(* IEC 61131-3 sources: elnaProjects/ElpcLogic/PomarKc7Unchanged/build_USO_ecl (part 2) *)

  (* OPC Init - AI. Стартовая инициализация тэгов _______________________________________________________*)

  (********************************************* Модуль A1-4 ******************************************************)

  AI_T_obmotki_fazy_1_k_HL       := ai.T_obmotki_fazy_1_k.HL;
  AI_T_obmotki_fazy_1_k_LL       := ai.T_obmotki_fazy_1_k.LL;
  AI_T_obmotki_fazy_1_k_newHL    := ai.T_obmotki_fazy_1_k.dHL;
  AI_T_obmotki_fazy_1_k_newLL    := ai.T_obmotki_fazy_1_k.dLL;

  AI_T_aktivnogo_zheleza_statora_1_k_HL        := ai.T_aktivnogo_zheleza_statora_1_k.HL;
  AI_T_aktivnogo_zheleza_statora_1_k_LL        := ai.T_aktivnogo_zheleza_statora_1_k.LL;
  AI_T_aktivnogo_zheleza_statora_1_k_newHL     := ai.T_aktivnogo_zheleza_statora_1_k.dHL;
  AI_T_aktivnogo_zheleza_statora_1_k_newLL     := ai.T_aktivnogo_zheleza_statora_1_k.dLL;

  AI_T_obmotki_fazy_2_k_HL	:= ai.T_obmotki_fazy_2_k.HL;
  AI_T_obmotki_fazy_2_k_LL	:= ai.T_obmotki_fazy_2_k.LL;
  AI_T_obmotki_fazy_2_k_newHL	:= ai.T_obmotki_fazy_2_k.dHL;
  AI_T_obmotki_fazy_2_k_newLL	:= ai.T_obmotki_fazy_2_k.dLL;

  AI_T_aktivnogo_zheleza_statora_2_k_HL       := ai.T_aktivnogo_zheleza_statora_2_k.HL;
  AI_T_aktivnogo_zheleza_statora_2_k_LL       := ai.T_aktivnogo_zheleza_statora_2_k.LL;
  AI_T_aktivnogo_zheleza_statora_2_k_newHL    := ai.T_aktivnogo_zheleza_statora_2_k.dHL;
  AI_T_aktivnogo_zheleza_statora_2_k_newLL    := ai.T_aktivnogo_zheleza_statora_2_k.dLL;

  AI_T_obmotki_fazy_3_k_HL	:= ai.T_obmotki_fazy_3_k.HL;
  AI_T_obmotki_fazy_3_k_LL	:= ai.T_obmotki_fazy_3_k.LL;
  AI_T_obmotki_fazy_3_k_newHL	:= ai.T_obmotki_fazy_3_k.dHL;
  AI_T_obmotki_fazy_3_k_newLL	:= ai.T_obmotki_fazy_3_k.dLL;

  AI_T_aktivnogo_zheleza_statora_3_k_HL	    := ai.T_aktivnogo_zheleza_statora_3_k.HL;
  AI_T_aktivnogo_zheleza_statora_3_k_LL	    := ai.T_aktivnogo_zheleza_statora_3_k.LL;
  AI_T_aktivnogo_zheleza_statora_3_k_newHL    := ai.T_aktivnogo_zheleza_statora_3_k.dHL;
  AI_T_aktivnogo_zheleza_statora_3_k_newLL    := ai.T_aktivnogo_zheleza_statora_3_k.dLL;

  AI_T_masla_v_maslobake_HL	:= ai.T_masla_v_maslobake.HL;
  AI_T_masla_v_maslobake_HW	:= ai.T_masla_v_maslobake.HW;
  AI_T_masla_v_maslobake_LL	:= ai.T_masla_v_maslobake.LL;
  AI_T_masla_v_maslobake_LW	:= ai.T_masla_v_maslobake.LW;
  AI_T_masla_v_maslobake_newHL	:= ai.T_masla_v_maslobake.dHL;
  AI_T_masla_v_maslobake_newHW	:= ai.T_masla_v_maslobake.dHW;
  AI_T_masla_v_maslobake_newLL	:= ai.T_masla_v_maslobake.dLL;
  AI_T_masla_v_maslobake_newLW	:= ai.T_masla_v_maslobake.dLW;

  (********************************************* Модуль A1-5 ******************************************************)
  AI_T_perednego_opornogo_podshipnika_dvigatelia_t1_HA	:= ai.T_perednego_opornogo_podshipnika_dvigatelia_t1.HA;
  AI_T_perednego_opornogo_podshipnika_dvigatelia_t1_HL	:= ai.T_perednego_opornogo_podshipnika_dvigatelia_t1.HL;
  AI_T_perednego_opornogo_podshipnika_dvigatelia_t1_HW	:= ai.T_perednego_opornogo_podshipnika_dvigatelia_t1.HW;
  AI_T_perednego_opornogo_podshipnika_dvigatelia_t1_LL	:= ai.T_perednego_opornogo_podshipnika_dvigatelia_t1.LL;
  AI_T_perednego_opornogo_podshipnika_dvigatelia_t1_newHA	:= ai.T_perednego_opornogo_podshipnika_dvigatelia_t1.dHA;
  AI_T_perednego_opornogo_podshipnika_dvigatelia_t1_newHW	:= ai.T_perednego_opornogo_podshipnika_dvigatelia_t1.dHW;
  AI_T_perednego_opornogo_podshipnika_dvigatelia_t1_newHL	:= ai.T_perednego_opornogo_podshipnika_dvigatelia_t1.dHL;
  AI_T_perednego_opornogo_podshipnika_dvigatelia_t1_newLL	:= ai.T_perednego_opornogo_podshipnika_dvigatelia_t1.dLL;

  AI_T_zadnego_opornogo_podshipnika_dvigatelia_t2_HA	:= ai.T_zadnego_opornogo_podshipnika_dvigatelia_t2.HA;
  AI_T_zadnego_opornogo_podshipnika_dvigatelia_t2_HL	:= ai.T_zadnego_opornogo_podshipnika_dvigatelia_t2.HL;
  AI_T_zadnego_opornogo_podshipnika_dvigatelia_t2_HW	:= ai.T_zadnego_opornogo_podshipnika_dvigatelia_t2.HW;
  AI_T_zadnego_opornogo_podshipnika_dvigatelia_t2_LL	:= ai.T_zadnego_opornogo_podshipnika_dvigatelia_t2.LL;
  AI_T_zadnego_opornogo_podshipnika_dvigatelia_t2_newHA	:= ai.T_zadnego_opornogo_podshipnika_dvigatelia_t2.dHA;
  AI_T_zadnego_opornogo_podshipnika_dvigatelia_t2_newHL	:= ai.T_zadnego_opornogo_podshipnika_dvigatelia_t2.dHL;
  AI_T_zadnego_opornogo_podshipnika_dvigatelia_t2_newHW	:= ai.T_zadnego_opornogo_podshipnika_dvigatelia_t2.dHW;
  AI_T_zadnego_opornogo_podshipnika_dvigatelia_t2_newLL	:= ai.T_zadnego_opornogo_podshipnika_dvigatelia_t2.dLL;

  AI_T_masla_na_slive_perednego_opornogo_podshipnika_dvigatelia_HL	:= ai.T_masla_na_slive_perednego_opornogo_podshipnika_dvigatelia.HL;
  AI_T_masla_na_slive_perednego_opornogo_podshipnika_dvigatelia_LL	:= ai.T_masla_na_slive_perednego_opornogo_podshipnika_dvigatelia.LL;
  AI_T_masla_na_slive_perednego_opornogo_podshipnika_dvigatelia_newHL	:= ai.T_masla_na_slive_perednego_opornogo_podshipnika_dvigatelia.dHL;
  AI_T_masla_na_slive_perednego_opornogo_podshipnika_dvigatelia_newLL	:= ai.T_masla_na_slive_perednego_opornogo_podshipnika_dvigatelia.dLL;

  AI_T_masla_na_slive_zadnego_opornogo_podshipnika_dvigatelia_HL	:= ai.T_masla_na_slive_zadnego_opornogo_podshipnika_dvigatelia.HL;
  AI_T_masla_na_slive_zadnego_opornogo_podshipnika_dvigatelia_LL	:= ai.T_masla_na_slive_zadnego_opornogo_podshipnika_dvigatelia.LL;
  AI_T_masla_na_slive_zadnego_opornogo_podshipnika_dvigatelia_newHL	:= ai.T_masla_na_slive_zadnego_opornogo_podshipnika_dvigatelia.dHL;
  AI_T_masla_na_slive_zadnego_opornogo_podshipnika_dvigatelia_newLL	:= ai.T_masla_na_slive_zadnego_opornogo_podshipnika_dvigatelia.dLL;

  AI_T_podshipnika_reduktora_t1_HA	:= ai.T_podshipnika_reduktora_t1.HA;
  AI_T_podshipnika_reduktora_t1_HL	:= ai.T_podshipnika_reduktora_t1.HL;
  AI_T_podshipnika_reduktora_t1_HW	:= ai.T_podshipnika_reduktora_t1.HW;
  AI_T_podshipnika_reduktora_t1_LL	:= ai.T_podshipnika_reduktora_t1.LL;
  AI_T_podshipnika_reduktora_t1_newHA	:= ai.T_podshipnika_reduktora_t1.dHA;
  AI_T_podshipnika_reduktora_t1_newHL	:= ai.T_podshipnika_reduktora_t1.dHL;
  AI_T_podshipnika_reduktora_t1_newHW	:= ai.T_podshipnika_reduktora_t1.dHW;
  AI_T_podshipnika_reduktora_t1_newLL	:= ai.T_podshipnika_reduktora_t1.dLL;

  AI_T_podshipnika_reduktora_t2_HA	:= ai.T_podshipnika_reduktora_t2.HA;
  AI_T_podshipnika_reduktora_t2_HL	:= ai.T_podshipnika_reduktora_t2.HL;
  AI_T_podshipnika_reduktora_t2_HW	:= ai.T_podshipnika_reduktora_t2.HW;
  AI_T_podshipnika_reduktora_t2_LL	:= ai.T_podshipnika_reduktora_t2.LL;
  AI_T_podshipnika_reduktora_t2_newHA	:= ai.T_podshipnika_reduktora_t2.dHA;
  AI_T_podshipnika_reduktora_t2_newHL	:= ai.T_podshipnika_reduktora_t2.dHL;
  AI_T_podshipnika_reduktora_t2_newHW	:= ai.T_podshipnika_reduktora_t2.dHW;
  AI_T_podshipnika_reduktora_t2_newLL	:= ai.T_podshipnika_reduktora_t2.dLL;

  AI_T_podshipnika_reduktora_t3_HA	:= ai.T_podshipnika_reduktora_t3.HA;
  AI_T_podshipnika_reduktora_t3_HL	:= ai.T_podshipnika_reduktora_t3.HL;
  AI_T_podshipnika_reduktora_t3_HW	:= ai.T_podshipnika_reduktora_t3.HW;
  AI_T_podshipnika_reduktora_t3_LL	:= ai.T_podshipnika_reduktora_t3.LL;
  AI_T_podshipnika_reduktora_t3_newHA	:= ai.T_podshipnika_reduktora_t3.dHA;
  AI_T_podshipnika_reduktora_t3_newHL	:= ai.T_podshipnika_reduktora_t3.dHL;
  AI_T_podshipnika_reduktora_t3_newHW	:= ai.T_podshipnika_reduktora_t3.dHW;
  AI_T_podshipnika_reduktora_t3_newLL	:= ai.T_podshipnika_reduktora_t3.dLL;

  AI_T_podshipnika_reduktora_t4_HA	:= ai.T_podshipnika_reduktora_t4.HA;
  AI_T_podshipnika_reduktora_t4_HL	:= ai.T_podshipnika_reduktora_t4.HL;
  AI_T_podshipnika_reduktora_t4_HW	:= ai.T_podshipnika_reduktora_t4.HW;
  AI_T_podshipnika_reduktora_t4_LL	:= ai.T_podshipnika_reduktora_t4.LL;
  AI_T_podshipnika_reduktora_t4_newHA	:= ai.T_podshipnika_reduktora_t4.dHA;
  AI_T_podshipnika_reduktora_t4_newHL	:= ai.T_podshipnika_reduktora_t4.dHL;
  AI_T_podshipnika_reduktora_t4_newHW	:= ai.T_podshipnika_reduktora_t4.dHW;
  AI_T_podshipnika_reduktora_t4_newLL	:= ai.T_podshipnika_reduktora_t4.dLL;

  (********************************************* Модуль A1-6 ******************************************************)

  AI_T_opornogo_podshipnika_nagnetatelia_t1_HA	:= ai.T_opornogo_podshipnika_nagnetatelia_t1.HA;
  AI_T_opornogo_podshipnika_nagnetatelia_t1_HL	:= ai.T_opornogo_podshipnika_nagnetatelia_t1.HL;
  AI_T_opornogo_podshipnika_nagnetatelia_t1_HW	:= ai.T_opornogo_podshipnika_nagnetatelia_t1.HW;
  AI_T_opornogo_podshipnika_nagnetatelia_t1_LL	:= ai.T_opornogo_podshipnika_nagnetatelia_t1.LL;
  AI_T_opornogo_podshipnika_nagnetatelia_t1_newHA	:= ai.T_opornogo_podshipnika_nagnetatelia_t1.dHA;
  AI_T_opornogo_podshipnika_nagnetatelia_t1_newHL	:= ai.T_opornogo_podshipnika_nagnetatelia_t1.dHL;
  AI_T_opornogo_podshipnika_nagnetatelia_t1_newHW	:= ai.T_opornogo_podshipnika_nagnetatelia_t1.dHW;
  AI_T_opornogo_podshipnika_nagnetatelia_t1_newLL	:= ai.T_opornogo_podshipnika_nagnetatelia_t1.dLL;

  AI_T_opornogo_podshipnika_nagnetatelia_t2_HA	:= ai.T_opornogo_podshipnika_nagnetatelia_t2.HA;
  AI_T_opornogo_podshipnika_nagnetatelia_t2_HL	:= ai.T_opornogo_podshipnika_nagnetatelia_t2.HL;
  AI_T_opornogo_podshipnika_nagnetatelia_t2_HW	:= ai.T_opornogo_podshipnika_nagnetatelia_t2.HW;
  AI_T_opornogo_podshipnika_nagnetatelia_t2_LL	:= ai.T_opornogo_podshipnika_nagnetatelia_t2.LL;
  AI_T_opornogo_podshipnika_nagnetatelia_t2_newHA	:= ai.T_opornogo_podshipnika_nagnetatelia_t2.dHA;
  AI_T_opornogo_podshipnika_nagnetatelia_t2_newHL	:= ai.T_opornogo_podshipnika_nagnetatelia_t2.dHL;
  AI_T_opornogo_podshipnika_nagnetatelia_t2_newHW	:= ai.T_opornogo_podshipnika_nagnetatelia_t2.dHW;
  AI_T_opornogo_podshipnika_nagnetatelia_t2_newLL	:= ai.T_opornogo_podshipnika_nagnetatelia_t2.dLL;

  AI_T_opornogo_podshipnika_nagnetatelia_t3_HA	:= ai.T_opornogo_podshipnika_nagnetatelia_t3.HA;
  AI_T_opornogo_podshipnika_nagnetatelia_t3_HL	:= ai.T_opornogo_podshipnika_nagnetatelia_t3.HL;
  AI_T_opornogo_podshipnika_nagnetatelia_t3_HW	:= ai.T_opornogo_podshipnika_nagnetatelia_t3.HW;
  AI_T_opornogo_podshipnika_nagnetatelia_t3_LL	:= ai.T_opornogo_podshipnika_nagnetatelia_t3.LL;
  AI_T_opornogo_podshipnika_nagnetatelia_t3_newHA	:= ai.T_opornogo_podshipnika_nagnetatelia_t3.dHA;
  AI_T_opornogo_podshipnika_nagnetatelia_t3_newHL	:= ai.T_opornogo_podshipnika_nagnetatelia_t3.dHL;
  AI_T_opornogo_podshipnika_nagnetatelia_t3_newHW	:= ai.T_opornogo_podshipnika_nagnetatelia_t3.dHW;
  AI_T_opornogo_podshipnika_nagnetatelia_t3_newLL	:= ai.T_opornogo_podshipnika_nagnetatelia_t3.dLL;

  AI_T_oporno_upornogo_podshipnika_nagnetatelia_t4_HA	:= ai.T_oporno_upornogo_podshipnika_nagnetatelia_t4.HA;
  AI_T_oporno_upornogo_podshipnika_nagnetatelia_t4_HL	:= ai.T_oporno_upornogo_podshipnika_nagnetatelia_t4.HL;
  AI_T_oporno_upornogo_podshipnika_nagnetatelia_t4_HW	:= ai.T_oporno_upornogo_podshipnika_nagnetatelia_t4.HW;
  AI_T_oporno_upornogo_podshipnika_nagnetatelia_t4_LL	:= ai.T_oporno_upornogo_podshipnika_nagnetatelia_t4.LL;
  AI_T_oporno_upornogo_podshipnika_nagnetatelia_t4_newHA	:= ai.T_oporno_upornogo_podshipnika_nagnetatelia_t4.dHA;
  AI_T_oporno_upornogo_podshipnika_nagnetatelia_t4_newHL	:= ai.T_oporno_upornogo_podshipnika_nagnetatelia_t4.dHL;
  AI_T_oporno_upornogo_podshipnika_nagnetatelia_t4_newHW	:= ai.T_oporno_upornogo_podshipnika_nagnetatelia_t4.dHW;
  AI_T_oporno_upornogo_podshipnika_nagnetatelia_t4_newLL	:= ai.T_oporno_upornogo_podshipnika_nagnetatelia_t4.dLL;

  AI_T_masla_do_AVOM_HL	:= ai.T_masla_do_AVOM.HL;
  AI_T_masla_do_AVOM_LL	:= ai.T_masla_do_AVOM.LL;
  AI_T_masla_do_AVOM_newHL	:= ai.T_masla_do_AVOM.dHL;
  AI_T_masla_do_AVOM_newLL	:= ai.T_masla_do_AVOM.dLL;

  AI_T_masla_posle_AVOM_HL	:= ai.T_masla_posle_AVOM.HL;
  AI_T_masla_posle_AVOM_LL	:= ai.T_masla_posle_AVOM.LL;
  AI_T_masla_posle_AVOM_newHL	:= ai.T_masla_posle_AVOM.dHL;
  AI_T_masla_posle_AVOM_newLL	:= ai.T_masla_posle_AVOM.dLL;

  AI_T_gaz_in_nagnetatelia_HL	          := ai.T_gaz_in_nagnetatelia.HL;
  AI_T_gaz_in_nagnetatelia_LL	          := ai.T_gaz_in_nagnetatelia.LL;
  AI_T_gaz_in_nagnetatelia_newHL	:= ai.T_gaz_in_nagnetatelia.dHL;
  AI_T_gaz_in_nagnetatelia_newLL	:= ai.T_gaz_in_nagnetatelia.dLL;

  AI_T_gaz_out_nagnetatelia_HA	          := ai.T_gaz_out_nagnetatelia.HA;
  AI_T_gaz_out_nagnetatelia_HL	          := ai.T_gaz_out_nagnetatelia.HL;
  AI_T_gaz_out_nagnetatelia_HW	          := ai.T_gaz_out_nagnetatelia.HW;
  AI_T_gaz_out_nagnetatelia_LL	          := ai.T_gaz_out_nagnetatelia.LL;
  AI_T_gaz_out_nagnetatelia_newHA	:= ai.T_gaz_out_nagnetatelia.dHA;
  AI_T_gaz_out_nagnetatelia_newHL	:= ai.T_gaz_out_nagnetatelia.dHL;
  AI_T_gaz_out_nagnetatelia_newHW	:= ai.T_gaz_out_nagnetatelia.dHW;
  AI_T_gaz_out_nagnetatelia_newLL	:= ai.T_gaz_out_nagnetatelia.dLL;

  (********************************************* Модуль A1-7 ******************************************************)

  AI_T_clodAir_dvigatelia_t1_HL	          := ai.T_clodAir_dvigatelia_t1.HL;
  AI_T_clodAir_dvigatelia_t1_LL	          := ai.T_clodAir_dvigatelia_t1.LL;
  AI_T_clodAir_dvigatelia_t1_newHL	:= ai.T_clodAir_dvigatelia_t1.dHL;
  AI_T_clodAir_dvigatelia_t1_newLL	:= ai.T_clodAir_dvigatelia_t1.dLL;

  AI_T_hotAir_dvigatelia_t1_HL	          := ai.T_hotAir_dvigatelia_t1.HL;
  AI_T_hotAir_dvigatelia_t1_LL	          := ai.T_hotAir_dvigatelia_t1.LL;
  AI_T_hotAir_dvigatelia_t1_newHL	:= ai.T_hotAir_dvigatelia_t1.dHL;
  AI_T_hotAir_dvigatelia_t1_newLL	:= ai.T_hotAir_dvigatelia_t1.dLL;

  (********************************************* Модуль A1-8 ******************************************************)

  AI_dPmaslo_gaz_HL	          := ai.dPmaslo_gaz.HL;
  AI_dPmaslo_gaz_LA	          := ai.dPmaslo_gaz.LA;
  AI_dPmaslo_gaz_LL	          := ai.dPmaslo_gaz.LL;
  AI_dPmaslo_gaz_LW	          := ai.dPmaslo_gaz.LW;
  AI_dPmaslo_gaz_newHL	:= ai.dPmaslo_gaz.dHL;
  AI_dPmaslo_gaz_newLA	:= ai.dPmaslo_gaz.dLA;
  AI_dPmaslo_gaz_newLL	:= ai.dPmaslo_gaz.dLL;
  AI_dPmaslo_gaz_newLW	:= ai.dPmaslo_gaz.dLW;
  AI_dPmaslo_gaz_newMaxChangeUP	 := ai.dPmaslo_gaz.dMaxChangeSpeed;
  AI_dPmaslo_gaz_newMaxChangeDown := ai.dPmaslo_gaz.dMaxChangeSpeedDown;

  AI_dP_gaza_na_konfuzore_nagnetatelia_HL	          := ai.dP_gaza_na_konfuzore_nagnetatelia.HL;
  AI_dP_gaza_na_konfuzore_nagnetatelia_LL	          := ai.dP_gaza_na_konfuzore_nagnetatelia.LL;
  AI_dP_gaza_na_konfuzore_nagnetatelia_newHL	:= ai.dP_gaza_na_konfuzore_nagnetatelia.dHL;
  AI_dP_gaza_na_konfuzore_nagnetatelia_newLL	:= ai.dP_gaza_na_konfuzore_nagnetatelia.dLL;

  AI_P_masla_uplotneniia_HL	:= ai.P_masla_uplotneniia.HL;
  AI_P_masla_uplotneniia_LL	:= ai.P_masla_uplotneniia.LL;
  AI_P_masla_uplotneniia_newHL	:= ai.P_masla_uplotneniia.dHL;
  AI_P_masla_uplotneniia_newLL	:= ai.P_masla_uplotneniia.dLL;

  AI_P_gaza_na_vkhode_nagnetatelia_HL	:= ai.P_gaza_na_vkhode_nagnetatelia.HL;
  AI_P_gaza_na_vkhode_nagnetatelia_LL	:= ai.P_gaza_na_vkhode_nagnetatelia.LL;
  AI_P_gaza_na_vkhode_nagnetatelia_newHL	:= ai.P_gaza_na_vkhode_nagnetatelia.dHL;
  AI_P_gaza_na_vkhode_nagnetatelia_newLL	:= ai.P_gaza_na_vkhode_nagnetatelia.dLL;

  AI_P_gaza_na_vykhode_nagnetatelia_HL	:= ai.P_gaza_na_vykhode_nagnetatelia.HL;
  AI_P_gaza_na_vykhode_nagnetatelia_LL	:= ai.P_gaza_na_vykhode_nagnetatelia.LL;
  AI_P_gaza_na_vykhode_nagnetatelia_newHL	:= ai.P_gaza_na_vykhode_nagnetatelia.dHL;
  AI_P_gaza_na_vykhode_nagnetatelia_newLL	:= ai.P_gaza_na_vykhode_nagnetatelia.dLL;

  AI_P_masla_smazki_nizkoe_HL	          := ai.P_masla_smazki_nizkoe.HL;
  AI_P_masla_smazki_nizkoe_LA	          := ai.P_masla_smazki_nizkoe.LA;
  AI_P_masla_smazki_nizkoe_LL	          := ai.P_masla_smazki_nizkoe.LL;
  AI_P_masla_smazki_nizkoe_LW	          := ai.P_masla_smazki_nizkoe.LW;
  AI_P_masla_smazki_nizkoe_newHL	:= ai.P_masla_smazki_nizkoe.dHL;
  AI_P_masla_smazki_nizkoe_newLA	:= ai.P_masla_smazki_nizkoe.dLA;
  AI_P_masla_smazki_nizkoe_newLL	:= ai.P_masla_smazki_nizkoe.dLL;
  AI_P_masla_smazki_nizkoe_newLW	:= ai.P_masla_smazki_nizkoe.dLW;

  AI_P_masla_smazki_srednee_posle_nasosov_HL	:= ai.P_masla_smazki_srednee_posle_nasosov.HL;
  AI_P_masla_smazki_srednee_posle_nasosov_LL	:= ai.P_masla_smazki_srednee_posle_nasosov.LL;
  AI_P_masla_smazki_srednee_posle_nasosov_LW	:= ai.P_masla_smazki_srednee_posle_nasosov.LW;
  AI_P_masla_smazki_srednee_posle_nasosov_newHL	:= ai.P_masla_smazki_srednee_posle_nasosov.dHL;
  AI_P_masla_smazki_srednee_posle_nasosov_newLL	:= ai.P_masla_smazki_srednee_posle_nasosov.dLL;
  AI_P_masla_smazki_srednee_posle_nasosov_newLW	:= ai.P_masla_smazki_srednee_posle_nasosov.dLW;

  (********************************************* Модуль A1-9 ******************************************************)

  AI_Vibratciia_STD_t1_HA	:= ai.Vibratciia_STD_t1.HA;
  AI_Vibratciia_STD_t1_HL	:= ai.Vibratciia_STD_t1.HL;
  AI_Vibratciia_STD_t1_HW	:= ai.Vibratciia_STD_t1.HW;
  AI_Vibratciia_STD_t1_LL	:= ai.Vibratciia_STD_t1.LL;
  AI_Vibratciia_STD_t1_newHA	:= ai.Vibratciia_STD_t1.dHA;
  AI_Vibratciia_STD_t1_newHL	:= ai.Vibratciia_STD_t1.dHL;
  AI_Vibratciia_STD_t1_newHW	:= ai.Vibratciia_STD_t1.dHW;
  AI_Vibratciia_STD_t1_newLL	:= ai.Vibratciia_STD_t1.dLL;

  AI_Vibratciia_STD_t2_HA	:= ai.Vibratciia_STD_t2.HA;
  AI_Vibratciia_STD_t2_HL	:= ai.Vibratciia_STD_t2.HL;
  AI_Vibratciia_STD_t2_HW	:= ai.Vibratciia_STD_t2.HW;
  AI_Vibratciia_STD_t2_LL	:= ai.Vibratciia_STD_t2.LL;
  AI_Vibratciia_STD_t2_newHA	:= ai.Vibratciia_STD_t2.dHA;
  AI_Vibratciia_STD_t2_newHL	:= ai.Vibratciia_STD_t2.dHL;
  AI_Vibratciia_STD_t2_newHW	:= ai.Vibratciia_STD_t2.dHW;
  AI_Vibratciia_STD_t2_newLL	:= ai.Vibratciia_STD_t2.dLL;

  AI_Vibratciia_rotora_nagnetatelia_t1_HA	          := ai.Vibratciia_rotora_nagnetatelia_t1.HA;
  AI_Vibratciia_rotora_nagnetatelia_t1_HL	          := ai.Vibratciia_rotora_nagnetatelia_t1.HL;
  AI_Vibratciia_rotora_nagnetatelia_t1_HW	          := ai.Vibratciia_rotora_nagnetatelia_t1.HW;
  AI_Vibratciia_rotora_nagnetatelia_t1_LL	          := ai.Vibratciia_rotora_nagnetatelia_t1.LL;
  AI_Vibratciia_rotora_nagnetatelia_t1_newHA	:= ai.Vibratciia_rotora_nagnetatelia_t1.dHA;
  AI_Vibratciia_rotora_nagnetatelia_t1_newHL	:= ai.Vibratciia_rotora_nagnetatelia_t1.dHL;
  AI_Vibratciia_rotora_nagnetatelia_t1_newHW	:= ai.Vibratciia_rotora_nagnetatelia_t1.dHW;
  AI_Vibratciia_rotora_nagnetatelia_t1_newLL	:= ai.Vibratciia_rotora_nagnetatelia_t1.dLL;

  AI_Vibratciia_rotora_nagnetatelia_t2_HA	          := ai.Vibratciia_rotora_nagnetatelia_t2.HA;
  AI_Vibratciia_rotora_nagnetatelia_t2_HL        	:= ai.Vibratciia_rotora_nagnetatelia_t2.HL;
  AI_Vibratciia_rotora_nagnetatelia_t2_HW    	:= ai.Vibratciia_rotora_nagnetatelia_t2.HW;
  AI_Vibratciia_rotora_nagnetatelia_t2_LL    	:= ai.Vibratciia_rotora_nagnetatelia_t2.LL;
  AI_Vibratciia_rotora_nagnetatelia_t2_newHA	:= ai.Vibratciia_rotora_nagnetatelia_t2.dHA;
  AI_Vibratciia_rotora_nagnetatelia_t2_newHL	:= ai.Vibratciia_rotora_nagnetatelia_t2.dHL;
  AI_Vibratciia_rotora_nagnetatelia_t2_newHW	:= ai.Vibratciia_rotora_nagnetatelia_t2.dHW;
  AI_Vibratciia_rotora_nagnetatelia_t2_newLL	:= ai.Vibratciia_rotora_nagnetatelia_t2.dLL;

  AI_Vibratciia_rotora_nagnetatelia_t3_HA    	:= ai.Vibratciia_rotora_nagnetatelia_t3.HA;
  AI_Vibratciia_rotora_nagnetatelia_t3_HL    	:= ai.Vibratciia_rotora_nagnetatelia_t3.HL;
  AI_Vibratciia_rotora_nagnetatelia_t3_HW    	:= ai.Vibratciia_rotora_nagnetatelia_t3.HW;
  AI_Vibratciia_rotora_nagnetatelia_t3_LL    	:= ai.Vibratciia_rotora_nagnetatelia_t3.LL;
  AI_Vibratciia_rotora_nagnetatelia_t3_newHA	:= ai.Vibratciia_rotora_nagnetatelia_t3.dHA;
  AI_Vibratciia_rotora_nagnetatelia_t3_newHL	:= ai.Vibratciia_rotora_nagnetatelia_t3.dHL;
  AI_Vibratciia_rotora_nagnetatelia_t3_newHW	:= ai.Vibratciia_rotora_nagnetatelia_t3.dHW;
  AI_Vibratciia_rotora_nagnetatelia_t3_newLL	:= ai.Vibratciia_rotora_nagnetatelia_t3.dLL;

  AI_Vibratciia_rotora_nagnetatelia_t4_HA    	:= ai.Vibratciia_rotora_nagnetatelia_t4.HA;
  AI_Vibratciia_rotora_nagnetatelia_t4_HL    	:= ai.Vibratciia_rotora_nagnetatelia_t4.HL;
  AI_Vibratciia_rotora_nagnetatelia_t4_HW    	:= ai.Vibratciia_rotora_nagnetatelia_t4.HW;
  AI_Vibratciia_rotora_nagnetatelia_t4_LL    	:= ai.Vibratciia_rotora_nagnetatelia_t4.LL;
  AI_Vibratciia_rotora_nagnetatelia_t4_newHA	:= ai.Vibratciia_rotora_nagnetatelia_t4.dHA;
  AI_Vibratciia_rotora_nagnetatelia_t4_newHL	:= ai.Vibratciia_rotora_nagnetatelia_t4.dHL;
  AI_Vibratciia_rotora_nagnetatelia_t4_newHW	:= ai.Vibratciia_rotora_nagnetatelia_t4.dHW;
  AI_Vibratciia_rotora_nagnetatelia_t4_newLL	:= ai.Vibratciia_rotora_nagnetatelia_t4.dLL;

  AI_Osevoi_sdvig_rotora_nagnetatelia_HA    	:= ai.Osevoi_sdvig_rotora_nagnetatelia.HA;
  AI_Osevoi_sdvig_rotora_nagnetatelia_HL    	:= ai.Osevoi_sdvig_rotora_nagnetatelia.HL;
  AI_Osevoi_sdvig_rotora_nagnetatelia_HW    	:= ai.Osevoi_sdvig_rotora_nagnetatelia.HW;
  AI_Osevoi_sdvig_rotora_nagnetatelia_LA    	:= ai.Osevoi_sdvig_rotora_nagnetatelia.LA;
  AI_Osevoi_sdvig_rotora_nagnetatelia_LL    	:= ai.Osevoi_sdvig_rotora_nagnetatelia.LL;
  AI_Osevoi_sdvig_rotora_nagnetatelia_LW    	:= ai.Osevoi_sdvig_rotora_nagnetatelia.LW;
  AI_Osevoi_sdvig_rotora_nagnetatelia_newHA	:= ai.Osevoi_sdvig_rotora_nagnetatelia.dHA;
  AI_Osevoi_sdvig_rotora_nagnetatelia_newHL	:= ai.Osevoi_sdvig_rotora_nagnetatelia.dHL;
  AI_Osevoi_sdvig_rotora_nagnetatelia_newHW	:= ai.Osevoi_sdvig_rotora_nagnetatelia.dHW;
  AI_Osevoi_sdvig_rotora_nagnetatelia_newLA	:= ai.Osevoi_sdvig_rotora_nagnetatelia.dLA;
  AI_Osevoi_sdvig_rotora_nagnetatelia_newLL	:= ai.Osevoi_sdvig_rotora_nagnetatelia.dLL;
  AI_Osevoi_sdvig_rotora_nagnetatelia_newLW	:= ai.Osevoi_sdvig_rotora_nagnetatelia.dLW;

  AI_Uroven_masla_v_maslobake_HL	:= ai.Uroven_masla_v_maslobake.HL;
  AI_Uroven_masla_v_maslobake_HW	:= ai.Uroven_masla_v_maslobake.HW;
  AI_Uroven_masla_v_maslobake_LA	:= ai.Uroven_masla_v_maslobake.LA;
  AI_Uroven_masla_v_maslobake_LL	:= ai.Uroven_masla_v_maslobake.LL;
  AI_Uroven_masla_v_maslobake_LW	:= ai.Uroven_masla_v_maslobake.LW;
  AI_Uroven_masla_v_maslobake_newHL	:= ai.Uroven_masla_v_maslobake.dHL;
  AI_Uroven_masla_v_maslobake_newHW	:= ai.Uroven_masla_v_maslobake.dHW;
  AI_Uroven_masla_v_maslobake_newLA	:= ai.Uroven_masla_v_maslobake.dLA;
  AI_Uroven_masla_v_maslobake_newLL	:= ai.Uroven_masla_v_maslobake.dLL;
  AI_Uroven_masla_v_maslobake_newLW	:= ai.Uroven_masla_v_maslobake.dLW;

  (********************************************* Модуль A1-10 ******************************************************)
  AI_T_vnytri_shkafa_HL	:= ai.T_vnytri_shkafa.HL;
  AI_T_vnytri_shkafa_LL	:= ai.T_vnytri_shkafa.LL;
  AI_T_vnytri_shkafa_HW	:= ai.T_vnytri_shkafa.HW;
  AI_T_vnytri_shkafa_LW	:= ai.T_vnytri_shkafa.LW;
  AI_T_vnytri_shkafa_newHL	:= ai.T_vnytri_shkafa.dHL;
  AI_T_vnytri_shkafa_newHW	:= ai.T_vnytri_shkafa.dHW;
  AI_T_vnytri_shkafa_newLL	:= ai.T_vnytri_shkafa.dLL;
  AI_T_vnytri_shkafa_newLW	:= ai.T_vnytri_shkafa.dLW;

  AI_Tok_vozbuzhdeniia_vozbuditelia_HL	:= ai.Tok_vozbuzhdeniia_vozbuditelia.HL;
  AI_Tok_vozbuzhdeniia_vozbuditelia_LL	:= ai.Tok_vozbuzhdeniia_vozbuditelia.LL;
  AI_Tok_vozbuzhdeniia_vozbuditelia_newHL	:= ai.Tok_vozbuzhdeniia_vozbuditelia.dHL;
  AI_Tok_vozbuzhdeniia_vozbuditelia_newLL	:= ai.Tok_vozbuzhdeniia_vozbuditelia.dLL;

  AI_Tok_statora_elektrodvigatelia_HL	:= ai.Tok_statora_elektrodvigatelia.HL;
  AI_Tok_statora_elektrodvigatelia_LL	:= ai.Tok_statora_elektrodvigatelia.LL;
  AI_Tok_statora_elektrodvigatelia_newHL	:= ai.Tok_statora_elektrodvigatelia.dHL;
  AI_Tok_statora_elektrodvigatelia_newLL	:= ai.Tok_statora_elektrodvigatelia.dLL;

  AI_Aktivnaia_moshchnost_HL	:= ai.Aktivnaia_moshchnost.HL;
  AI_Aktivnaia_moshchnost_LL	:= ai.Aktivnaia_moshchnost.LL;
  AI_Aktivnaia_moshchnost_newHL	:= ai.Aktivnaia_moshchnost.dHL;
  AI_Aktivnaia_moshchnost_newLL	:= ai.Aktivnaia_moshchnost.dLL;

  AI_Reaktivnaia_moshchnost_HL    	:= ai.Reaktivnaia_moshchnost.HL;
  AI_Reaktivnaia_moshchnost_LL    	:= ai.Reaktivnaia_moshchnost.LL;
  AI_Reaktivnaia_moshchnost_newHL	:= ai.Reaktivnaia_moshchnost.dHL;
  AI_Reaktivnaia_moshchnost_newLL	:= ai.Reaktivnaia_moshchnost.dLL;

  AI_VoltageSHU_osnovnoi_vvod_HL	:= ai.VoltageSHU_osnovnoi_vvod.HL;
  AI_VoltageSHU_osnovnoi_vvod_HW	:= ai.VoltageSHU_osnovnoi_vvod.HW;
  AI_VoltageSHU_osnovnoi_vvod_LL	:= ai.VoltageSHU_osnovnoi_vvod.LL;
  AI_VoltageSHU_osnovnoi_vvod_LW	:= ai.VoltageSHU_osnovnoi_vvod.LW;
  AI_VoltageSHU_osnovnoi_vvod_newHL	:= ai.VoltageSHU_osnovnoi_vvod.dHL;
  AI_VoltageSHU_osnovnoi_vvod_newHW	:= ai.VoltageSHU_osnovnoi_vvod.dHW;
  AI_VoltageSHU_osnovnoi_vvod_newLL	:= ai.VoltageSHU_osnovnoi_vvod.dLL;
  AI_VoltageSHU_osnovnoi_vvod_newLW	:= ai.VoltageSHU_osnovnoi_vvod.dLW;

  AI_VoltageSHU_rezervnyi_vvod_HL	:= ai.VoltageSHU_rezervnyi_vvod.HL;
  AI_VoltageSHU_rezervnyi_vvod_HW	:= ai.VoltageSHU_rezervnyi_vvod.HW;
  AI_VoltageSHU_rezervnyi_vvod_LL	:= ai.VoltageSHU_rezervnyi_vvod.LL;
  AI_VoltageSHU_rezervnyi_vvod_LW	:= ai.VoltageSHU_rezervnyi_vvod.LW;
  AI_VoltageSHU_rezervnyi_vvod_newHL	:= ai.VoltageSHU_rezervnyi_vvod.dHL;
  AI_VoltageSHU_rezervnyi_vvod_newHW	:= ai.VoltageSHU_rezervnyi_vvod.dHW;
  AI_VoltageSHU_rezervnyi_vvod_newLL	:= ai.VoltageSHU_rezervnyi_vvod.dLL;
  AI_VoltageSHU_rezervnyi_vvod_newLW	:= ai.VoltageSHU_rezervnyi_vvod.dLW;
END_FUNCTION_BLOCK

FUNCTION_BLOCK OPC_AI_get
  VAR_EXTERNAL
    ai : AiConfig;
    AI_Aktivnaia_moshchnost_HL : LREAL;
    AI_Aktivnaia_moshchnost_LL : LREAL;
    AI_Aktivnaia_moshchnost_command : UINT;
    AI_Aktivnaia_moshchnost_newHL : LREAL;
    AI_Aktivnaia_moshchnost_newLL : LREAL;
    AI_Aktivnaia_moshchnost_status : UDINT;
    AI_Aktivnaia_moshchnost_value : LREAL;
    AI_Osevoi_sdvig_rotora_nagnetatelia_HA : LREAL;
    AI_Osevoi_sdvig_rotora_nagnetatelia_HL : LREAL;
    AI_Osevoi_sdvig_rotora_nagnetatelia_HW : LREAL;
    AI_Osevoi_sdvig_rotora_nagnetatelia_LA : LREAL;
    AI_Osevoi_sdvig_rotora_nagnetatelia_LL : LREAL;
    AI_Osevoi_sdvig_rotora_nagnetatelia_LW : LREAL;
    AI_Osevoi_sdvig_rotora_nagnetatelia_command : UINT;
    AI_Osevoi_sdvig_rotora_nagnetatelia_newHA : LREAL;
    AI_Osevoi_sdvig_rotora_nagnetatelia_newHL : LREAL;
    AI_Osevoi_sdvig_rotora_nagnetatelia_newHW : LREAL;
    AI_Osevoi_sdvig_rotora_nagnetatelia_newLA : LREAL;
    AI_Osevoi_sdvig_rotora_nagnetatelia_newLL : LREAL;
    AI_Osevoi_sdvig_rotora_nagnetatelia_newLW : LREAL;
    AI_Osevoi_sdvig_rotora_nagnetatelia_status : UDINT;
    AI_Osevoi_sdvig_rotora_nagnetatelia_value : LREAL;
    AI_P_gaza_na_vkhode_nagnetatelia_HL : LREAL;
    AI_P_gaza_na_vkhode_nagnetatelia_LL : LREAL;
    AI_P_gaza_na_vkhode_nagnetatelia_command : UINT;
    AI_P_gaza_na_vkhode_nagnetatelia_newHL : LREAL;
    AI_P_gaza_na_vkhode_nagnetatelia_newLL : LREAL;
    AI_P_gaza_na_vkhode_nagnetatelia_status : UDINT;
    AI_P_gaza_na_vkhode_nagnetatelia_value : LREAL;
    AI_P_gaza_na_vykhode_nagnetatelia_HL : LREAL;
    AI_P_gaza_na_vykhode_nagnetatelia_LL : LREAL;
    AI_P_gaza_na_vykhode_nagnetatelia_command : UINT;
    AI_P_gaza_na_vykhode_nagnetatelia_newHL : LREAL;
    AI_P_gaza_na_vykhode_nagnetatelia_newLL : LREAL;
    AI_P_gaza_na_vykhode_nagnetatelia_status : UDINT;
    AI_P_gaza_na_vykhode_nagnetatelia_value : LREAL;
    AI_P_masla_smazki_nizkoe_HL : LREAL;
    AI_P_masla_smazki_nizkoe_LA : LREAL;
    AI_P_masla_smazki_nizkoe_LL : LREAL;
    AI_P_masla_smazki_nizkoe_LW : LREAL;
    AI_P_masla_smazki_nizkoe_command : UINT;
    AI_P_masla_smazki_nizkoe_newHL : LREAL;
    AI_P_masla_smazki_nizkoe_newLA : LREAL;
    AI_P_masla_smazki_nizkoe_newLL : LREAL;
    AI_P_masla_smazki_nizkoe_newLW : LREAL;
    AI_P_masla_smazki_nizkoe_status : UDINT;
    AI_P_masla_smazki_nizkoe_value : LREAL;
    AI_P_masla_smazki_srednee_posle_nasosov_HL : LREAL;
    AI_P_masla_smazki_srednee_posle_nasosov_LL : LREAL;
    AI_P_masla_smazki_srednee_posle_nasosov_LW : LREAL;
    AI_P_masla_smazki_srednee_posle_nasosov_command : UINT;
    AI_P_masla_smazki_srednee_posle_nasosov_newHL : LREAL;
    AI_P_masla_smazki_srednee_posle_nasosov_newLL : LREAL;
    AI_P_masla_smazki_srednee_posle_nasosov_newLW : LREAL;
    AI_P_masla_smazki_srednee_posle_nasosov_status : UDINT;
    AI_P_masla_smazki_srednee_posle_nasosov_value : LREAL;
    AI_P_masla_uplotneniia_HL : LREAL;
    AI_P_masla_uplotneniia_LL : LREAL;
    AI_P_masla_uplotneniia_command : UINT;
    AI_P_masla_uplotneniia_newHL : LREAL;
    AI_P_masla_uplotneniia_newLL : LREAL;
    AI_P_masla_uplotneniia_status : UDINT;
    AI_P_masla_uplotneniia_value : LREAL;
    AI_Reaktivnaia_moshchnost_HL : LREAL;
    AI_Reaktivnaia_moshchnost_LL : LREAL;
    AI_Reaktivnaia_moshchnost_command : UINT;
    AI_Reaktivnaia_moshchnost_newHL : LREAL;
    AI_Reaktivnaia_moshchnost_newLL : LREAL;
    AI_Reaktivnaia_moshchnost_status : UDINT;
    AI_Reaktivnaia_moshchnost_value : LREAL;
    AI_T_aktivnogo_zheleza_statora_1_k_HL : LREAL;
    AI_T_aktivnogo_zheleza_statora_1_k_LL : LREAL;
    AI_T_aktivnogo_zheleza_statora_1_k_command : UINT;
    AI_T_aktivnogo_zheleza_statora_1_k_newHL : LREAL;
    AI_T_aktivnogo_zheleza_statora_1_k_newLL : LREAL;
    AI_T_aktivnogo_zheleza_statora_1_k_status : UDINT;
    AI_T_aktivnogo_zheleza_statora_1_k_value : LREAL;
    AI_T_aktivnogo_zheleza_statora_2_k_HL : LREAL;
    AI_T_aktivnogo_zheleza_statora_2_k_LL : LREAL;
    AI_T_aktivnogo_zheleza_statora_2_k_command : UINT;
    AI_T_aktivnogo_zheleza_statora_2_k_newHL : LREAL;
    AI_T_aktivnogo_zheleza_statora_2_k_newLL : LREAL;
    AI_T_aktivnogo_zheleza_statora_2_k_status : UDINT;
    AI_T_aktivnogo_zheleza_statora_2_k_value : LREAL;
    AI_T_aktivnogo_zheleza_statora_3_k_HL : LREAL;
    AI_T_aktivnogo_zheleza_statora_3_k_LL : LREAL;
    AI_T_aktivnogo_zheleza_statora_3_k_command : UINT;
    AI_T_aktivnogo_zheleza_statora_3_k_newHL : LREAL;
    AI_T_aktivnogo_zheleza_statora_3_k_newLL : LREAL;
    AI_T_aktivnogo_zheleza_statora_3_k_status : UDINT;
    AI_T_aktivnogo_zheleza_statora_3_k_value : LREAL;
    AI_T_clodAir_dvigatelia_t1_HL : LREAL;
    AI_T_clodAir_dvigatelia_t1_LL : LREAL;
    AI_T_clodAir_dvigatelia_t1_command : UINT;
    AI_T_clodAir_dvigatelia_t1_newHL : LREAL;
    AI_T_clodAir_dvigatelia_t1_newLL : LREAL;
    AI_T_clodAir_dvigatelia_t1_status : UDINT;
    AI_T_clodAir_dvigatelia_t1_value : LREAL;
    AI_T_gaz_in_nagnetatelia_HL : LREAL;
    AI_T_gaz_in_nagnetatelia_LL : LREAL;
    AI_T_gaz_in_nagnetatelia_command : UINT;
    AI_T_gaz_in_nagnetatelia_newHL : LREAL;
    AI_T_gaz_in_nagnetatelia_newLL : LREAL;
    AI_T_gaz_in_nagnetatelia_status : UDINT;
    AI_T_gaz_in_nagnetatelia_value : LREAL;
    AI_T_gaz_out_nagnetatelia_HL : LREAL;
    AI_T_gaz_out_nagnetatelia_LL : LREAL;
    AI_T_gaz_out_nagnetatelia_command : UINT;
    AI_T_gaz_out_nagnetatelia_newHL : LREAL;
    AI_T_gaz_out_nagnetatelia_newLL : LREAL;
    AI_T_gaz_out_nagnetatelia_status : UDINT;
    AI_T_gaz_out_nagnetatelia_value : LREAL;
    AI_T_hotAir_dvigatelia_t1_HL : LREAL;
    AI_T_hotAir_dvigatelia_t1_LL : LREAL;
    AI_T_hotAir_dvigatelia_t1_command : UINT;
    AI_T_hotAir_dvigatelia_t1_newHL : LREAL;
    AI_T_hotAir_dvigatelia_t1_newLL : LREAL;
    AI_T_hotAir_dvigatelia_t1_status : UDINT;
    AI_T_hotAir_dvigatelia_t1_value : LREAL;
    AI_T_masla_do_AVOM_HL : LREAL;
    AI_T_masla_do_AVOM_LL : LREAL;
    AI_T_masla_do_AVOM_command : UINT;
    AI_T_masla_do_AVOM_newHL : LREAL;
    AI_T_masla_do_AVOM_newLL : LREAL;
    AI_T_masla_do_AVOM_status : UDINT;
    AI_T_masla_do_AVOM_value : LREAL;
    AI_T_masla_na_slive_perednego_opornogo_podshipnika_dvigatelia_HL : LREAL;
    AI_T_masla_na_slive_perednego_opornogo_podshipnika_dvigatelia_LL : LREAL;
    AI_T_masla_na_slive_perednego_opornogo_podshipnika_dvigatelia_command : UINT;
    AI_T_masla_na_slive_perednego_opornogo_podshipnika_dvigatelia_newHL : LREAL;
    AI_T_masla_na_slive_perednego_opornogo_podshipnika_dvigatelia_newLL : LREAL;
    AI_T_masla_na_slive_perednego_opornogo_podshipnika_dvigatelia_status : UDINT;
    AI_T_masla_na_slive_perednego_opornogo_podshipnika_dvigatelia_value : LREAL;
    AI_T_masla_na_slive_zadnego_opornogo_podshipnika_dvigatelia_HL : LREAL;
    AI_T_masla_na_slive_zadnego_opornogo_podshipnika_dvigatelia_LL : LREAL;
    AI_T_masla_na_slive_zadnego_opornogo_podshipnika_dvigatelia_command : UINT;
    AI_T_masla_na_slive_zadnego_opornogo_podshipnika_dvigatelia_newHL : LREAL;
    AI_T_masla_na_slive_zadnego_opornogo_podshipnika_dvigatelia_newLL : LREAL;
    AI_T_masla_na_slive_zadnego_opornogo_podshipnika_dvigatelia_status : UDINT;
    AI_T_masla_na_slive_zadnego_opornogo_podshipnika_dvigatelia_value : LREAL;
    AI_T_masla_posle_AVOM_HL : LREAL;
    AI_T_masla_posle_AVOM_LL : LREAL;
    AI_T_masla_posle_AVOM_command : UINT;
    AI_T_masla_posle_AVOM_newHL : LREAL;
    AI_T_masla_posle_AVOM_newLL : LREAL;
    AI_T_masla_posle_AVOM_status : UDINT;
    AI_T_masla_posle_AVOM_value : LREAL;
    AI_T_masla_v_maslobake_HL : LREAL;
    AI_T_masla_v_maslobake_HW : LREAL;
    AI_T_masla_v_maslobake_LL : LREAL;
    AI_T_masla_v_maslobake_LW : LREAL;
    AI_T_masla_v_maslobake_command : UINT;
    AI_T_masla_v_maslobake_newHL : LREAL;
    AI_T_masla_v_maslobake_newHW : LREAL;
    AI_T_masla_v_maslobake_newLL : LREAL;
    AI_T_masla_v_maslobake_newLW : LREAL;
    AI_T_masla_v_maslobake_status : UDINT;
    AI_T_masla_v_maslobake_value : LREAL;
    AI_T_obmotki_fazy_1_k_HL : LREAL;
    AI_T_obmotki_fazy_1_k_LL : LREAL;
    AI_T_obmotki_fazy_1_k_command : UINT;
    AI_T_obmotki_fazy_1_k_newHL : LREAL;
    AI_T_obmotki_fazy_1_k_newLL : LREAL;
    AI_T_obmotki_fazy_1_k_status : UDINT;
    AI_T_obmotki_fazy_1_k_value : LREAL;
    AI_T_obmotki_fazy_2_k_HL : LREAL;
    AI_T_obmotki_fazy_2_k_LL : LREAL;
    AI_T_obmotki_fazy_2_k_command : UINT;
    AI_T_obmotki_fazy_2_k_newHL : LREAL;
    AI_T_obmotki_fazy_2_k_newLL : LREAL;
    AI_T_obmotki_fazy_2_k_status : UDINT;
    AI_T_obmotki_fazy_2_k_value : LREAL;
    AI_T_obmotki_fazy_3_k_HL : LREAL;
    AI_T_obmotki_fazy_3_k_LL : LREAL;
    AI_T_obmotki_fazy_3_k_command : UINT;
    AI_T_obmotki_fazy_3_k_newHL : LREAL;
    AI_T_obmotki_fazy_3_k_newLL : LREAL;
    AI_T_obmotki_fazy_3_k_status : UDINT;
    AI_T_obmotki_fazy_3_k_value : LREAL;
    AI_T_oporno_upornogo_podshipnika_nagnetatelia_t4_HA : LREAL;
    AI_T_oporno_upornogo_podshipnika_nagnetatelia_t4_HL : LREAL;
    AI_T_oporno_upornogo_podshipnika_nagnetatelia_t4_HW : LREAL;
    AI_T_oporno_upornogo_podshipnika_nagnetatelia_t4_LL : LREAL;
    AI_T_oporno_upornogo_podshipnika_nagnetatelia_t4_command : UINT;
    AI_T_oporno_upornogo_podshipnika_nagnetatelia_t4_newHA : LREAL;
    AI_T_oporno_upornogo_podshipnika_nagnetatelia_t4_newHL : LREAL;
    AI_T_oporno_upornogo_podshipnika_nagnetatelia_t4_newHW : LREAL;
    AI_T_oporno_upornogo_podshipnika_nagnetatelia_t4_newLL : LREAL;
    AI_T_oporno_upornogo_podshipnika_nagnetatelia_t4_status : UDINT;
    AI_T_oporno_upornogo_podshipnika_nagnetatelia_t4_value : LREAL;
    AI_T_opornogo_podshipnika_nagnetatelia_t1_HA : LREAL;
    AI_T_opornogo_podshipnika_nagnetatelia_t1_HL : LREAL;
    AI_T_opornogo_podshipnika_nagnetatelia_t1_HW : LREAL;
    AI_T_opornogo_podshipnika_nagnetatelia_t1_LL : LREAL;
    AI_T_opornogo_podshipnika_nagnetatelia_t1_command : UINT;
    AI_T_opornogo_podshipnika_nagnetatelia_t1_newHA : LREAL;
    AI_T_opornogo_podshipnika_nagnetatelia_t1_newHL : LREAL;
    AI_T_opornogo_podshipnika_nagnetatelia_t1_newHW : LREAL;
    AI_T_opornogo_podshipnika_nagnetatelia_t1_newLL : LREAL;
    AI_T_opornogo_podshipnika_nagnetatelia_t1_status : UDINT;
    AI_T_opornogo_podshipnika_nagnetatelia_t1_value : LREAL;
    AI_T_opornogo_podshipnika_nagnetatelia_t2_HA : LREAL;
    AI_T_opornogo_podshipnika_nagnetatelia_t2_HL : LREAL;
    AI_T_opornogo_podshipnika_nagnetatelia_t2_HW : LREAL;
    AI_T_opornogo_podshipnika_nagnetatelia_t2_LL : LREAL;
    AI_T_opornogo_podshipnika_nagnetatelia_t2_command : UINT;
    AI_T_opornogo_podshipnika_nagnetatelia_t2_newHA : LREAL;
    AI_T_opornogo_podshipnika_nagnetatelia_t2_newHL : LREAL;
    AI_T_opornogo_podshipnika_nagnetatelia_t2_newHW : LREAL;
    AI_T_opornogo_podshipnika_nagnetatelia_t2_newLL : LREAL;
    AI_T_opornogo_podshipnika_nagnetatelia_t2_status : UDINT;
    AI_T_opornogo_podshipnika_nagnetatelia_t2_value : LREAL;
    AI_T_opornogo_podshipnika_nagnetatelia_t3_HA : LREAL;
    AI_T_opornogo_podshipnika_nagnetatelia_t3_HL : LREAL;
    AI_T_opornogo_podshipnika_nagnetatelia_t3_HW : LREAL;
    AI_T_opornogo_podshipnika_nagnetatelia_t3_LL : LREAL;
    AI_T_opornogo_podshipnika_nagnetatelia_t3_command : UINT;
    AI_T_opornogo_podshipnika_nagnetatelia_t3_newHA : LREAL;
    AI_T_opornogo_podshipnika_nagnetatelia_t3_newHL : LREAL;
    AI_T_opornogo_podshipnika_nagnetatelia_t3_newHW : LREAL;
    AI_T_opornogo_podshipnika_nagnetatelia_t3_newLL : LREAL;
    AI_T_opornogo_podshipnika_nagnetatelia_t3_status : UDINT;
    AI_T_opornogo_podshipnika_nagnetatelia_t3_value : LREAL;
    AI_T_perednego_opornogo_podshipnika_dvigatelia_t1_HL : LREAL;
    AI_T_perednego_opornogo_podshipnika_dvigatelia_t1_LL : LREAL;
    AI_T_perednego_opornogo_podshipnika_dvigatelia_t1_command : UINT;
    AI_T_perednego_opornogo_podshipnika_dvigatelia_t1_newHL : LREAL;
    AI_T_perednego_opornogo_podshipnika_dvigatelia_t1_newLL : LREAL;
    AI_T_perednego_opornogo_podshipnika_dvigatelia_t1_status : UDINT;
    AI_T_perednego_opornogo_podshipnika_dvigatelia_t1_value : LREAL;
    AI_T_podshipnika_reduktora_t1_HA : LREAL;
    AI_T_podshipnika_reduktora_t1_HL : LREAL;
    AI_T_podshipnika_reduktora_t1_HW : LREAL;
    AI_T_podshipnika_reduktora_t1_LL : LREAL;
    AI_T_podshipnika_reduktora_t1_command : UINT;
    AI_T_podshipnika_reduktora_t1_newHA : LREAL;
    AI_T_podshipnika_reduktora_t1_newHL : LREAL;
    AI_T_podshipnika_reduktora_t1_newHW : LREAL;
    AI_T_podshipnika_reduktora_t1_newLL : LREAL;
    AI_T_podshipnika_reduktora_t1_status : UDINT;
    AI_T_podshipnika_reduktora_t1_value : LREAL;
    AI_T_podshipnika_reduktora_t2_HA : LREAL;
    AI_T_podshipnika_reduktora_t2_HL : LREAL;
    AI_T_podshipnika_reduktora_t2_HW : LREAL;
    AI_T_podshipnika_reduktora_t2_LL : LREAL;
    AI_T_podshipnika_reduktora_t2_command : UINT;
    AI_T_podshipnika_reduktora_t2_newHA : LREAL;
    AI_T_podshipnika_reduktora_t2_newHL : LREAL;
    AI_T_podshipnika_reduktora_t2_newHW : LREAL;
    AI_T_podshipnika_reduktora_t2_newLL : LREAL;
    AI_T_podshipnika_reduktora_t2_status : UDINT;
    AI_T_podshipnika_reduktora_t2_value : LREAL;
    AI_T_podshipnika_reduktora_t3_HA : LREAL;
    AI_T_podshipnika_reduktora_t3_HL : LREAL;
    AI_T_podshipnika_reduktora_t3_HW : LREAL;
    AI_T_podshipnika_reduktora_t3_LL : LREAL;
    AI_T_podshipnika_reduktora_t3_command : UINT;
    AI_T_podshipnika_reduktora_t3_newHA : LREAL;
    AI_T_podshipnika_reduktora_t3_newHL : LREAL;
    AI_T_podshipnika_reduktora_t3_newHW : LREAL;
    AI_T_podshipnika_reduktora_t3_newLL : LREAL;
    AI_T_podshipnika_reduktora_t3_status : UDINT;
    AI_T_podshipnika_reduktora_t3_value : LREAL;
    AI_T_podshipnika_reduktora_t4_HA : LREAL;
    AI_T_podshipnika_reduktora_t4_HL : LREAL;
    AI_T_podshipnika_reduktora_t4_HW : LREAL;
    AI_T_podshipnika_reduktora_t4_LL : LREAL;
    AI_T_podshipnika_reduktora_t4_command : UINT;
    AI_T_podshipnika_reduktora_t4_newHA : LREAL;
    AI_T_podshipnika_reduktora_t4_newHL : LREAL;
    AI_T_podshipnika_reduktora_t4_newHW : LREAL;
    AI_T_podshipnika_reduktora_t4_newLL : LREAL;
    AI_T_podshipnika_reduktora_t4_status : UDINT;
    AI_T_podshipnika_reduktora_t4_value : LREAL;
    AI_T_zadnego_opornogo_podshipnika_dvigatelia_t2_HA : LREAL;
    AI_T_zadnego_opornogo_podshipnika_dvigatelia_t2_HL : LREAL;
    AI_T_zadnego_opornogo_podshipnika_dvigatelia_t2_HW : LREAL;
    AI_T_zadnego_opornogo_podshipnika_dvigatelia_t2_LL : LREAL;
    AI_T_zadnego_opornogo_podshipnika_dvigatelia_t2_command : UINT;
    AI_T_zadnego_opornogo_podshipnika_dvigatelia_t2_newHA : LREAL;
    AI_T_zadnego_opornogo_podshipnika_dvigatelia_t2_newHL : LREAL;
    AI_T_zadnego_opornogo_podshipnika_dvigatelia_t2_newHW : LREAL;
    AI_T_zadnego_opornogo_podshipnika_dvigatelia_t2_newLL : LREAL;
    AI_T_zadnego_opornogo_podshipnika_dvigatelia_t2_status : UDINT;
    AI_T_zadnego_opornogo_podshipnika_dvigatelia_t2_value : LREAL;
    AI_Tok_statora_elektrodvigatelia_HL : LREAL;
    AI_Tok_statora_elektrodvigatelia_LL : LREAL;
    AI_Tok_statora_elektrodvigatelia_command : UINT;
    AI_Tok_statora_elektrodvigatelia_newHL : LREAL;
    AI_Tok_statora_elektrodvigatelia_newLL : LREAL;
    AI_Tok_statora_elektrodvigatelia_status : UDINT;
    AI_Tok_statora_elektrodvigatelia_value : LREAL;
    AI_Tok_vozbuzhdeniia_vozbuditelia_HL : LREAL;
    AI_Tok_vozbuzhdeniia_vozbuditelia_LL : LREAL;
    AI_Tok_vozbuzhdeniia_vozbuditelia_command : UINT;
    AI_Tok_vozbuzhdeniia_vozbuditelia_newHL : LREAL;
    AI_Tok_vozbuzhdeniia_vozbuditelia_newLL : LREAL;
    AI_Tok_vozbuzhdeniia_vozbuditelia_status : UDINT;
    AI_Tok_vozbuzhdeniia_vozbuditelia_value : LREAL;
    AI_Uroven_masla_v_maslobake_HL : LREAL;
    AI_Uroven_masla_v_maslobake_HW : LREAL;
    AI_Uroven_masla_v_maslobake_LA : LREAL;
    AI_Uroven_masla_v_maslobake_LL : LREAL;
    AI_Uroven_masla_v_maslobake_LW : LREAL;
    AI_Uroven_masla_v_maslobake_command : UINT;
    AI_Uroven_masla_v_maslobake_newHL : LREAL;
    AI_Uroven_masla_v_maslobake_newHW : LREAL;
    AI_Uroven_masla_v_maslobake_newLA : LREAL;
    AI_Uroven_masla_v_maslobake_newLL : LREAL;
    AI_Uroven_masla_v_maslobake_newLW : LREAL;
    AI_Uroven_masla_v_maslobake_status : UDINT;
    AI_Uroven_masla_v_maslobake_value : LREAL;
    AI_Vibratciia_STD_t1_HA : LREAL;
    AI_Vibratciia_STD_t1_HL : LREAL;
    AI_Vibratciia_STD_t1_HW : LREAL;
    AI_Vibratciia_STD_t1_LL : LREAL;
    AI_Vibratciia_STD_t1_command : UINT;
    AI_Vibratciia_STD_t1_newHA : LREAL;
    AI_Vibratciia_STD_t1_newHL : LREAL;
    AI_Vibratciia_STD_t1_newHW : LREAL;
    AI_Vibratciia_STD_t1_newLL : LREAL;
    AI_Vibratciia_STD_t1_status : UDINT;
    AI_Vibratciia_STD_t1_value : LREAL;
    AI_Vibratciia_STD_t2_HA : LREAL;
    AI_Vibratciia_STD_t2_HL : LREAL;
    AI_Vibratciia_STD_t2_HW : LREAL;
    AI_Vibratciia_STD_t2_LL : LREAL;
    AI_Vibratciia_STD_t2_command : UINT;
    AI_Vibratciia_STD_t2_newHA : LREAL;
    AI_Vibratciia_STD_t2_newHL : LREAL;
    AI_Vibratciia_STD_t2_newHW : LREAL;
    AI_Vibratciia_STD_t2_newLL : LREAL;
    AI_Vibratciia_STD_t2_status : UDINT;
    AI_Vibratciia_STD_t2_value : LREAL;
    AI_Vibratciia_rotora_nagnetatelia_t1_HA : LREAL;
    AI_Vibratciia_rotora_nagnetatelia_t1_HL : LREAL;
    AI_Vibratciia_rotora_nagnetatelia_t1_HW : LREAL;
    AI_Vibratciia_rotora_nagnetatelia_t1_LL : LREAL;
    AI_Vibratciia_rotora_nagnetatelia_t1_command : UINT;
    AI_Vibratciia_rotora_nagnetatelia_t1_newHA : LREAL;
    AI_Vibratciia_rotora_nagnetatelia_t1_newHL : LREAL;
    AI_Vibratciia_rotora_nagnetatelia_t1_newHW : LREAL;
    AI_Vibratciia_rotora_nagnetatelia_t1_newLL : LREAL;
    AI_Vibratciia_rotora_nagnetatelia_t1_status : UDINT;
    AI_Vibratciia_rotora_nagnetatelia_t1_value : LREAL;
    AI_Vibratciia_rotora_nagnetatelia_t2_HA : LREAL;
    AI_Vibratciia_rotora_nagnetatelia_t2_HL : LREAL;
    AI_Vibratciia_rotora_nagnetatelia_t2_HW : LREAL;
    AI_Vibratciia_rotora_nagnetatelia_t2_LL : LREAL;
    AI_Vibratciia_rotora_nagnetatelia_t2_command : UINT;
    AI_Vibratciia_rotora_nagnetatelia_t2_newHA : LREAL;
    AI_Vibratciia_rotora_nagnetatelia_t2_newHL : LREAL;
    AI_Vibratciia_rotora_nagnetatelia_t2_newHW : LREAL;
    AI_Vibratciia_rotora_nagnetatelia_t2_newLL : LREAL;
    AI_Vibratciia_rotora_nagnetatelia_t2_status : UDINT;
    AI_Vibratciia_rotora_nagnetatelia_t2_value : LREAL;
    AI_Vibratciia_rotora_nagnetatelia_t3_HA : LREAL;
    AI_Vibratciia_rotora_nagnetatelia_t3_HL : LREAL;
    AI_Vibratciia_rotora_nagnetatelia_t3_HW : LREAL;
    AI_Vibratciia_rotora_nagnetatelia_t3_LL : LREAL;
    AI_Vibratciia_rotora_nagnetatelia_t3_command : UINT;
    AI_Vibratciia_rotora_nagnetatelia_t3_newHA : LREAL;
    AI_Vibratciia_rotora_nagnetatelia_t3_newHL : LREAL;
    AI_Vibratciia_rotora_nagnetatelia_t3_newHW : LREAL;
    AI_Vibratciia_rotora_nagnetatelia_t3_newLL : LREAL;
    AI_Vibratciia_rotora_nagnetatelia_t3_status : UDINT;
    AI_Vibratciia_rotora_nagnetatelia_t3_value : LREAL;
    AI_Vibratciia_rotora_nagnetatelia_t4_HA : LREAL;
    AI_Vibratciia_rotora_nagnetatelia_t4_HL : LREAL;
    AI_Vibratciia_rotora_nagnetatelia_t4_HW : LREAL;
    AI_Vibratciia_rotora_nagnetatelia_t4_LL : LREAL;
    AI_Vibratciia_rotora_nagnetatelia_t4_command : UINT;
    AI_Vibratciia_rotora_nagnetatelia_t4_newHA : LREAL;
    AI_Vibratciia_rotora_nagnetatelia_t4_newHL : LREAL;
    AI_Vibratciia_rotora_nagnetatelia_t4_newHW : LREAL;
    AI_Vibratciia_rotora_nagnetatelia_t4_newLL : LREAL;
    AI_Vibratciia_rotora_nagnetatelia_t4_status : UDINT;
    AI_Vibratciia_rotora_nagnetatelia_t4_value : LREAL;
    AI_VoltageSHU_osnovnoi_vvod_HL : LREAL;
    AI_VoltageSHU_osnovnoi_vvod_HW : LREAL;
    AI_VoltageSHU_osnovnoi_vvod_LL : LREAL;
    AI_VoltageSHU_osnovnoi_vvod_LW : LREAL;
    AI_VoltageSHU_osnovnoi_vvod_command : UINT;
    AI_VoltageSHU_osnovnoi_vvod_newHL : LREAL;
    AI_VoltageSHU_osnovnoi_vvod_newHW : LREAL;
    AI_VoltageSHU_osnovnoi_vvod_newLL : LREAL;
    AI_VoltageSHU_osnovnoi_vvod_newLW : LREAL;
    AI_VoltageSHU_osnovnoi_vvod_status : UDINT;
    AI_VoltageSHU_osnovnoi_vvod_value : LREAL;
    AI_VoltageSHU_rezervnyi_vvod_HL : LREAL;
    AI_VoltageSHU_rezervnyi_vvod_HW : LREAL;
    AI_VoltageSHU_rezervnyi_vvod_LL : LREAL;
    AI_VoltageSHU_rezervnyi_vvod_LW : LREAL;
    AI_VoltageSHU_rezervnyi_vvod_command : UINT;
    AI_VoltageSHU_rezervnyi_vvod_newHL : LREAL;
    AI_VoltageSHU_rezervnyi_vvod_newHW : LREAL;
    AI_VoltageSHU_rezervnyi_vvod_newLL : LREAL;
    AI_VoltageSHU_rezervnyi_vvod_newLW : LREAL;
    AI_VoltageSHU_rezervnyi_vvod_status : UDINT;
    AI_VoltageSHU_rezervnyi_vvod_value : LREAL;
    AI_dP_gaza_na_konfuzore_nagnetatelia_HL : LREAL;
    AI_dP_gaza_na_konfuzore_nagnetatelia_LL : LREAL;
    AI_dP_gaza_na_konfuzore_nagnetatelia_command : UINT;
    AI_dP_gaza_na_konfuzore_nagnetatelia_newHL : LREAL;
    AI_dP_gaza_na_konfuzore_nagnetatelia_newLL : LREAL;
    AI_dP_gaza_na_konfuzore_nagnetatelia_status : UDINT;
    AI_dP_gaza_na_konfuzore_nagnetatelia_value : LREAL;
    AI_dPmaslo_gaz_HL : LREAL;
    AI_dPmaslo_gaz_LA : LREAL;
    AI_dPmaslo_gaz_LL : LREAL;
    AI_dPmaslo_gaz_LW : LREAL;
    AI_dPmaslo_gaz_command : UINT;
    AI_dPmaslo_gaz_newHL : LREAL;
    AI_dPmaslo_gaz_newLA : LREAL;
    AI_dPmaslo_gaz_newLL : LREAL;
    AI_dPmaslo_gaz_newLW : LREAL;
    AI_dPmaslo_gaz_status : UDINT;
    AI_dPmaslo_gaz_value : LREAL;
    AI_T_perednego_opornogo_podshipnika_dvigatelia_t1_HA : LREAL;
    AI_T_perednego_opornogo_podshipnika_dvigatelia_t1_HW : LREAL;
    AI_T_perednego_opornogo_podshipnika_dvigatelia_t1_newHA : LREAL;
    AI_T_perednego_opornogo_podshipnika_dvigatelia_t1_newHW : LREAL;
    AI_T_gaz_out_nagnetatelia_HA : LREAL;
    AI_T_gaz_out_nagnetatelia_HW : LREAL;
    AI_T_gaz_out_nagnetatelia_newHA : LREAL;
    AI_T_gaz_out_nagnetatelia_newHW : LREAL;
    AI_T_vnytri_shkafa_command : UINT;
    AI_T_vnytri_shkafa_newHL : LREAL;
    AI_T_vnytri_shkafa_newHW : LREAL;
    AI_T_vnytri_shkafa_newLL : LREAL;
    AI_T_vnytri_shkafa_newLW : LREAL;
    AI_dPmaslo_gaz_newMaxChangeDown : LREAL;
    AI_dPmaslo_gaz_newMaxChangeUP : LREAL;
  END_VAR

  (* OPC Get - AI. Чтение текущих состояний тэгов _______________________________________________________*)

  (********************************************* Модуль A1-4 ******************************************************)

   ai.T_obmotki_fazy_1_k.inCommand_ARM	:= UINT_TO_WORD(AI_T_obmotki_fazy_1_k_command);
   ai.T_obmotki_fazy_1_k.dHL    	:= AI_T_obmotki_fazy_1_k_newHL;
   ai.T_obmotki_fazy_1_k.dLL    	:= AI_T_obmotki_fazy_1_k_newLL;

   ai.T_aktivnogo_zheleza_statora_1_k.inCommand_ARM	:= UINT_TO_WORD(AI_T_aktivnogo_zheleza_statora_1_k_command);
   ai.T_aktivnogo_zheleza_statora_1_k.dHL    	:= AI_T_aktivnogo_zheleza_statora_1_k_newHL;
   ai.T_aktivnogo_zheleza_statora_1_k.dLL    	:= AI_T_aktivnogo_zheleza_statora_1_k_newLL;

   ai.T_obmotki_fazy_2_k.inCommand_ARM	:= UINT_TO_WORD(AI_T_obmotki_fazy_2_k_command);
   ai.T_obmotki_fazy_2_k.dHL    	:= AI_T_obmotki_fazy_2_k_newHL;
   ai.T_obmotki_fazy_2_k.dLL    	:= AI_T_obmotki_fazy_2_k_newLL;

   ai.T_aktivnogo_zheleza_statora_2_k.inCommand_ARM	:= UINT_TO_WORD(AI_T_aktivnogo_zheleza_statora_2_k_command);
   ai.T_aktivnogo_zheleza_statora_2_k.dHL    	:= AI_T_aktivnogo_zheleza_statora_2_k_newHL;
   ai.T_aktivnogo_zheleza_statora_2_k.dLL    	:= AI_T_aktivnogo_zheleza_statora_2_k_newLL;

   ai.T_obmotki_fazy_3_k.inCommand_ARM	:= UINT_TO_WORD(AI_T_obmotki_fazy_3_k_command);
   ai.T_obmotki_fazy_3_k.dHL    	:= AI_T_obmotki_fazy_3_k_newHL;
   ai.T_obmotki_fazy_3_k.dLL    	:= AI_T_obmotki_fazy_3_k_newLL;

   ai.T_aktivnogo_zheleza_statora_3_k.inCommand_ARM	:= UINT_TO_WORD(AI_T_aktivnogo_zheleza_statora_3_k_command);
   ai.T_aktivnogo_zheleza_statora_3_k.dHL    	:= AI_T_aktivnogo_zheleza_statora_3_k_newHL;
   ai.T_aktivnogo_zheleza_statora_3_k.dLL    	:= AI_T_aktivnogo_zheleza_statora_3_k_newLL;

   ai.T_masla_v_maslobake.inCommand_ARM	:= UINT_TO_WORD(AI_T_masla_v_maslobake_command);
   ai.T_masla_v_maslobake.dHL    	:= AI_T_masla_v_maslobake_newHL;
   ai.T_masla_v_maslobake.dHW    	:= AI_T_masla_v_maslobake_newHW;
   ai.T_masla_v_maslobake.dLL    	:= AI_T_masla_v_maslobake_newLL;
   ai.T_masla_v_maslobake.dLW    	:= AI_T_masla_v_maslobake_newLW;

  (********************************************* Модуль A1-5 ******************************************************)

   ai.T_perednego_opornogo_podshipnika_dvigatelia_t1.inCommand_ARM	:= UINT_TO_WORD(AI_T_perednego_opornogo_podshipnika_dvigatelia_t1_command);
   ai.T_perednego_opornogo_podshipnika_dvigatelia_t1.dHA        	:= AI_T_perednego_opornogo_podshipnika_dvigatelia_t1_newHA;
   ai.T_perednego_opornogo_podshipnika_dvigatelia_t1.dHL        	:= AI_T_perednego_opornogo_podshipnika_dvigatelia_t1_newHL;
   ai.T_perednego_opornogo_podshipnika_dvigatelia_t1.dHW        	:= AI_T_perednego_opornogo_podshipnika_dvigatelia_t1_newHW;
   ai.T_perednego_opornogo_podshipnika_dvigatelia_t1.dLL        	:= AI_T_perednego_opornogo_podshipnika_dvigatelia_t1_newLL;

   ai.T_zadnego_opornogo_podshipnika_dvigatelia_t2.inCommand_ARM	:= UINT_TO_WORD(AI_T_zadnego_opornogo_podshipnika_dvigatelia_t2_command);
   ai.T_zadnego_opornogo_podshipnika_dvigatelia_t2.dHA        	:= AI_T_zadnego_opornogo_podshipnika_dvigatelia_t2_newHA;
   ai.T_zadnego_opornogo_podshipnika_dvigatelia_t2.dHL        	:= AI_T_zadnego_opornogo_podshipnika_dvigatelia_t2_newHL;
   ai.T_zadnego_opornogo_podshipnika_dvigatelia_t2.dHW        	:= AI_T_zadnego_opornogo_podshipnika_dvigatelia_t2_newHW;
   ai.T_zadnego_opornogo_podshipnika_dvigatelia_t2.dLL        	:= AI_T_zadnego_opornogo_podshipnika_dvigatelia_t2_newLL;

   ai.T_masla_na_slive_perednego_opornogo_podshipnika_dvigatelia.inCommand_ARM	:= UINT_TO_WORD(AI_T_masla_na_slive_perednego_opornogo_podshipnika_dvigatelia_command);
   ai.T_masla_na_slive_perednego_opornogo_podshipnika_dvigatelia.dHL    	:= AI_T_masla_na_slive_perednego_opornogo_podshipnika_dvigatelia_newHL;
   ai.T_masla_na_slive_perednego_opornogo_podshipnika_dvigatelia.dLL    	:= AI_T_masla_na_slive_perednego_opornogo_podshipnika_dvigatelia_newLL;

   ai.T_masla_na_slive_zadnego_opornogo_podshipnika_dvigatelia.inCommand_ARM	:= UINT_TO_WORD(AI_T_masla_na_slive_zadnego_opornogo_podshipnika_dvigatelia_command);
   ai.T_masla_na_slive_zadnego_opornogo_podshipnika_dvigatelia.dHL        	:= AI_T_masla_na_slive_zadnego_opornogo_podshipnika_dvigatelia_newHL;
   ai.T_masla_na_slive_zadnego_opornogo_podshipnika_dvigatelia.dLL        	:= AI_T_masla_na_slive_zadnego_opornogo_podshipnika_dvigatelia_newLL;

  ai.T_podshipnika_reduktora_t1.inCommand_ARM	:= UINT_TO_WORD(AI_T_podshipnika_reduktora_t1_command);
   ai.T_podshipnika_reduktora_t1.dHA	:= AI_T_podshipnika_reduktora_t1_newHA;
   ai.T_podshipnika_reduktora_t1.dHL	:= AI_T_podshipnika_reduktora_t1_newHL;
   ai.T_podshipnika_reduktora_t1.dHW	:= AI_T_podshipnika_reduktora_t1_newHW;
   ai.T_podshipnika_reduktora_t1.dLL	:= AI_T_podshipnika_reduktora_t1_newLL;

   ai.T_podshipnika_reduktora_t2.inCommand_ARM	:= UINT_TO_WORD(AI_T_podshipnika_reduktora_t2_command);
   ai.T_podshipnika_reduktora_t2.dHA	:= AI_T_podshipnika_reduktora_t2_newHA;
   ai.T_podshipnika_reduktora_t2.dHL	:= AI_T_podshipnika_reduktora_t2_newHL;
   ai.T_podshipnika_reduktora_t2.dHW	:= AI_T_podshipnika_reduktora_t2_newHW;
   ai.T_podshipnika_reduktora_t2.dLL	:= AI_T_podshipnika_reduktora_t2_newLL;

   ai.T_podshipnika_reduktora_t3.inCommand_ARM	:= UINT_TO_WORD(AI_T_podshipnika_reduktora_t3_command);
   ai.T_podshipnika_reduktora_t3.dHA	:= AI_T_podshipnika_reduktora_t3_newHA;
   ai.T_podshipnika_reduktora_t3.dHL	:= AI_T_podshipnika_reduktora_t3_newHL;
   ai.T_podshipnika_reduktora_t3.dHW	:= AI_T_podshipnika_reduktora_t3_newHW;
   ai.T_podshipnika_reduktora_t3.dLL	:= AI_T_podshipnika_reduktora_t3_newLL;

   ai.T_podshipnika_reduktora_t4.inCommand_ARM	:= UINT_TO_WORD(AI_T_podshipnika_reduktora_t4_command);
   ai.T_podshipnika_reduktora_t4.dHA	:= AI_T_podshipnika_reduktora_t4_newHA;
   ai.T_podshipnika_reduktora_t4.dHL	:= AI_T_podshipnika_reduktora_t4_newHL;
   ai.T_podshipnika_reduktora_t4.dHW	:= AI_T_podshipnika_reduktora_t4_newHW;
   ai.T_podshipnika_reduktora_t4.dLL	:= AI_T_podshipnika_reduktora_t4_newLL;

  (********************************************* Модуль A1-6 ******************************************************)

  ai.T_opornogo_podshipnika_nagnetatelia_t1.inCommand_ARM	:= UINT_TO_WORD(AI_T_opornogo_podshipnika_nagnetatelia_t1_command);
   ai.T_opornogo_podshipnika_nagnetatelia_t1.dHA    	:= AI_T_opornogo_podshipnika_nagnetatelia_t1_newHA;
   ai.T_opornogo_podshipnika_nagnetatelia_t1.dHL    	:= AI_T_opornogo_podshipnika_nagnetatelia_t1_newHL;
   ai.T_opornogo_podshipnika_nagnetatelia_t1.dHW    	:= AI_T_opornogo_podshipnika_nagnetatelia_t1_newHW;
   ai.T_opornogo_podshipnika_nagnetatelia_t1.dLL    	:= AI_T_opornogo_podshipnika_nagnetatelia_t1_newLL;

   ai.T_opornogo_podshipnika_nagnetatelia_t2.inCommand_ARM	:= UINT_TO_WORD(AI_T_opornogo_podshipnika_nagnetatelia_t2_command);
   ai.T_opornogo_podshipnika_nagnetatelia_t2.dHA    	:= AI_T_opornogo_podshipnika_nagnetatelia_t2_newHA;
   ai.T_opornogo_podshipnika_nagnetatelia_t2.dHL    	:= AI_T_opornogo_podshipnika_nagnetatelia_t2_newHL;
   ai.T_opornogo_podshipnika_nagnetatelia_t2.dHW    	:= AI_T_opornogo_podshipnika_nagnetatelia_t2_newHW;
   ai.T_opornogo_podshipnika_nagnetatelia_t2.dLL    	:= AI_T_opornogo_podshipnika_nagnetatelia_t2_newLL;

   ai.T_opornogo_podshipnika_nagnetatelia_t3.inCommand_ARM	:= UINT_TO_WORD(AI_T_opornogo_podshipnika_nagnetatelia_t3_command);
   ai.T_opornogo_podshipnika_nagnetatelia_t3.dHA            	:= AI_T_opornogo_podshipnika_nagnetatelia_t3_newHA;
   ai.T_opornogo_podshipnika_nagnetatelia_t3.dHL    	:= AI_T_opornogo_podshipnika_nagnetatelia_t3_newHL;
   ai.T_opornogo_podshipnika_nagnetatelia_t3.dHW    	:= AI_T_opornogo_podshipnika_nagnetatelia_t3_newHW;
   ai.T_opornogo_podshipnika_nagnetatelia_t3.dLL    	:= AI_T_opornogo_podshipnika_nagnetatelia_t3_newLL;

   ai.T_oporno_upornogo_podshipnika_nagnetatelia_t4.inCommand_ARM	:= UINT_TO_WORD(AI_T_oporno_upornogo_podshipnika_nagnetatelia_t4_command);
   ai.T_oporno_upornogo_podshipnika_nagnetatelia_t4.dHA        	:= AI_T_oporno_upornogo_podshipnika_nagnetatelia_t4_newHA;
   ai.T_oporno_upornogo_podshipnika_nagnetatelia_t4.dHL        	:= AI_T_oporno_upornogo_podshipnika_nagnetatelia_t4_newHL;
   ai.T_oporno_upornogo_podshipnika_nagnetatelia_t4.dHW        	:= AI_T_oporno_upornogo_podshipnika_nagnetatelia_t4_newHW;
   ai.T_oporno_upornogo_podshipnika_nagnetatelia_t4.dLL        	:= AI_T_oporno_upornogo_podshipnika_nagnetatelia_t4_newLL;

   ai.T_masla_do_AVOM.inCommand_ARM	:= UINT_TO_WORD(AI_T_masla_do_AVOM_command);
   ai.T_masla_do_AVOM.dHL        	:= AI_T_masla_do_AVOM_newHL;
   ai.T_masla_do_AVOM.dLL        	:= AI_T_masla_do_AVOM_newLL;

   ai.T_masla_posle_AVOM.inCommand_ARM	:= UINT_TO_WORD(AI_T_masla_posle_AVOM_command);
   ai.T_masla_posle_AVOM.dHL    	:= AI_T_masla_posle_AVOM_newHL;
   ai.T_masla_posle_AVOM.dLL    	:= AI_T_masla_posle_AVOM_newLL;

   ai.T_gaz_in_nagnetatelia.inCommand_ARM	:= UINT_TO_WORD(AI_T_gaz_in_nagnetatelia_command);
   ai.T_gaz_in_nagnetatelia.dHL    	:= AI_T_gaz_in_nagnetatelia_newHL;
   ai.T_gaz_in_nagnetatelia.dLL    	:= AI_T_gaz_in_nagnetatelia_newLL;

   ai.T_gaz_out_nagnetatelia.inCommand_ARM    := UINT_TO_WORD(AI_T_gaz_out_nagnetatelia_command);
   ai.T_gaz_out_nagnetatelia.dHA              := AI_T_gaz_out_nagnetatelia_newHA;
   ai.T_gaz_out_nagnetatelia.dHL              := AI_T_gaz_out_nagnetatelia_newHL;
   ai.T_gaz_out_nagnetatelia.dHW              := AI_T_gaz_out_nagnetatelia_newHW;
   ai.T_gaz_out_nagnetatelia.dLL              := AI_T_gaz_out_nagnetatelia_newLL;

  (********************************************* Модуль A1-7 ******************************************************)

   ai.T_clodAir_dvigatelia_t1.inCommand_ARM	:= UINT_TO_WORD(AI_T_clodAir_dvigatelia_t1_command);
   ai.T_clodAir_dvigatelia_t1.dHL            	:= AI_T_clodAir_dvigatelia_t1_newHL;
   ai.T_clodAir_dvigatelia_t1.dLL            	:= AI_T_clodAir_dvigatelia_t1_newLL;

   ai.T_hotAir_dvigatelia_t1.inCommand_ARM	:= UINT_TO_WORD(AI_T_hotAir_dvigatelia_t1_command);
   ai.T_hotAir_dvigatelia_t1.dHL            	:= AI_T_hotAir_dvigatelia_t1_newHL;
   ai.T_hotAir_dvigatelia_t1.dLL            	:= AI_T_hotAir_dvigatelia_t1_newLL;

  (********************************************* Модуль A1-8 ******************************************************)

   ai.dPmaslo_gaz.inCommand_ARM	:= UINT_TO_WORD(AI_dPmaslo_gaz_command);
   ai.dPmaslo_gaz.dHL    	:= AI_dPmaslo_gaz_newHL;
   ai.dPmaslo_gaz.dLA    	:= AI_dPmaslo_gaz_newLA;
   ai.dPmaslo_gaz.dLL    	:= AI_dPmaslo_gaz_newLL;
   ai.dPmaslo_gaz.dLW    	:= AI_dPmaslo_gaz_newLW;
   ai.dPmaslo_gaz.dMaxChangeSpeed 	:= AI_dPmaslo_gaz_newMaxChangeUP;
   ai.dPmaslo_gaz.dMaxChangeSpeedDown     := AI_dPmaslo_gaz_newMaxChangeDown;

   ai.dP_gaza_na_konfuzore_nagnetatelia.inCommand_ARM	:= UINT_TO_WORD(AI_dP_gaza_na_konfuzore_nagnetatelia_command);
   ai.dP_gaza_na_konfuzore_nagnetatelia.dHL            	:= AI_dP_gaza_na_konfuzore_nagnetatelia_newHL;
   ai.dP_gaza_na_konfuzore_nagnetatelia.dLL            	:= AI_dP_gaza_na_konfuzore_nagnetatelia_newLL;

   ai.P_masla_uplotneniia.inCommand_ARM	:= UINT_TO_WORD(AI_P_masla_uplotneniia_command);
   ai.P_masla_uplotneniia.dHL    	:= AI_P_masla_uplotneniia_newHL;
   ai.P_masla_uplotneniia.dLL    	:= AI_P_masla_uplotneniia_newLL;

   ai.P_gaza_na_vkhode_nagnetatelia.inCommand_ARM	:= UINT_TO_WORD(AI_P_gaza_na_vkhode_nagnetatelia_command);
   ai.P_gaza_na_vkhode_nagnetatelia.dHL    	:= AI_P_gaza_na_vkhode_nagnetatelia_newHL;
   ai.P_gaza_na_vkhode_nagnetatelia.dLL    	:= AI_P_gaza_na_vkhode_nagnetatelia_newLL;

   ai.P_gaza_na_vykhode_nagnetatelia.inCommand_ARM	:= UINT_TO_WORD(AI_P_gaza_na_vykhode_nagnetatelia_command);
   ai.P_gaza_na_vykhode_nagnetatelia.dHL    	:= AI_P_gaza_na_vykhode_nagnetatelia_newHL;
   ai.P_gaza_na_vykhode_nagnetatelia.dLL    	:= AI_P_gaza_na_vykhode_nagnetatelia_newLL;

  ai.P_masla_smazki_nizkoe.inCommand_ARM	:= UINT_TO_WORD(AI_P_masla_smazki_nizkoe_command);
   ai.P_masla_smazki_nizkoe.dHL    	:= AI_P_masla_smazki_nizkoe_newHL;
   ai.P_masla_smazki_nizkoe.dLA    	:= AI_P_masla_smazki_nizkoe_newLA;
   ai.P_masla_smazki_nizkoe.dLL    	:= AI_P_masla_smazki_nizkoe_newLL;
   ai.P_masla_smazki_nizkoe.dLW    	:= AI_P_masla_smazki_nizkoe_newLW;

   ai.P_masla_smazki_srednee_posle_nasosov.inCommand_ARM	:= UINT_TO_WORD(AI_P_masla_smazki_srednee_posle_nasosov_command);
   ai.P_masla_smazki_srednee_posle_nasosov.dHL        	:= AI_P_masla_smazki_srednee_posle_nasosov_newHL;
   ai.P_masla_smazki_srednee_posle_nasosov.dLL        	:= AI_P_masla_smazki_srednee_posle_nasosov_newLL;
   ai.P_masla_smazki_srednee_posle_nasosov.dLW        	:= AI_P_masla_smazki_srednee_posle_nasosov_newLW;

  (********************************************* Модуль A1-9 ******************************************************)

  ai.Vibratciia_STD_t1.inCommand_ARM	:= UINT_TO_WORD(AI_Vibratciia_STD_t1_command);
   ai.Vibratciia_STD_t1.dHA        	:= AI_Vibratciia_STD_t1_newHA;
   ai.Vibratciia_STD_t1.dHL        	:= AI_Vibratciia_STD_t1_newHL;
   ai.Vibratciia_STD_t1.dHW        	:= AI_Vibratciia_STD_t1_newHW;
   ai.Vibratciia_STD_t1.dLL        	:= AI_Vibratciia_STD_t1_newLL;

   ai.Vibratciia_STD_t2.inCommand_ARM	:= UINT_TO_WORD(AI_Vibratciia_STD_t2_command);
   ai.Vibratciia_STD_t2.dHA        	:= AI_Vibratciia_STD_t2_newHA;
   ai.Vibratciia_STD_t2.dHL        	:= AI_Vibratciia_STD_t2_newHL;
   ai.Vibratciia_STD_t2.dHW        	:= AI_Vibratciia_STD_t2_newHW;
   ai.Vibratciia_STD_t2.dLL        	:= AI_Vibratciia_STD_t2_newLL;

  ai.Vibratciia_rotora_nagnetatelia_t1.inCommand_ARM    := UINT_TO_WORD(AI_Vibratciia_rotora_nagnetatelia_t1_command);
   ai.Vibratciia_rotora_nagnetatelia_t1.dHA             := AI_Vibratciia_rotora_nagnetatelia_t1_newHA;
   ai.Vibratciia_rotora_nagnetatelia_t1.dHL             := AI_Vibratciia_rotora_nagnetatelia_t1_newHL;
   ai.Vibratciia_rotora_nagnetatelia_t1.dHW             := AI_Vibratciia_rotora_nagnetatelia_t1_newHW;
   ai.Vibratciia_rotora_nagnetatelia_t1.dLL             := AI_Vibratciia_rotora_nagnetatelia_t1_newLL;

   ai.Vibratciia_rotora_nagnetatelia_t2.inCommand_ARM    := UINT_TO_WORD(AI_Vibratciia_rotora_nagnetatelia_t2_command);
   ai.Vibratciia_rotora_nagnetatelia_t2.dHA	     := AI_Vibratciia_rotora_nagnetatelia_t2_newHA;
   ai.Vibratciia_rotora_nagnetatelia_t2.dHL              := AI_Vibratciia_rotora_nagnetatelia_t2_newHL;
   ai.Vibratciia_rotora_nagnetatelia_t2.dHW	     := AI_Vibratciia_rotora_nagnetatelia_t2_newHW;
   ai.Vibratciia_rotora_nagnetatelia_t2.dLL	     := AI_Vibratciia_rotora_nagnetatelia_t2_newLL;

   ai.Vibratciia_rotora_nagnetatelia_t3.inCommand_ARM    := UINT_TO_WORD(AI_Vibratciia_rotora_nagnetatelia_t3_command);
   ai.Vibratciia_rotora_nagnetatelia_t3.dHA	     := AI_Vibratciia_rotora_nagnetatelia_t3_newHA;
   ai.Vibratciia_rotora_nagnetatelia_t3.dHL	     := AI_Vibratciia_rotora_nagnetatelia_t3_newHL;
   ai.Vibratciia_rotora_nagnetatelia_t3.dHW	     := AI_Vibratciia_rotora_nagnetatelia_t3_newHW;
   ai.Vibratciia_rotora_nagnetatelia_t3.dLL	     := AI_Vibratciia_rotora_nagnetatelia_t3_newLL;

   ai.Vibratciia_rotora_nagnetatelia_t4.inCommand_ARM    := UINT_TO_WORD(AI_Vibratciia_rotora_nagnetatelia_t4_command);
   ai.Vibratciia_rotora_nagnetatelia_t4.dHA	     := AI_Vibratciia_rotora_nagnetatelia_t4_newHA;
   ai.Vibratciia_rotora_nagnetatelia_t4.dHL	     := AI_Vibratciia_rotora_nagnetatelia_t4_newHL;
   ai.Vibratciia_rotora_nagnetatelia_t4.dHW	     := AI_Vibratciia_rotora_nagnetatelia_t4_newHW;
   ai.Vibratciia_rotora_nagnetatelia_t4.dLL	     := AI_Vibratciia_rotora_nagnetatelia_t4_newLL;

   ai.Osevoi_sdvig_rotora_nagnetatelia.inCommand_ARM    := UINT_TO_WORD(AI_Osevoi_sdvig_rotora_nagnetatelia_command);
   ai.Osevoi_sdvig_rotora_nagnetatelia.dHA	    := AI_Osevoi_sdvig_rotora_nagnetatelia_newHA;
   ai.Osevoi_sdvig_rotora_nagnetatelia.dHL	    := AI_Osevoi_sdvig_rotora_nagnetatelia_newHL;
   ai.Osevoi_sdvig_rotora_nagnetatelia.dHW	    := AI_Osevoi_sdvig_rotora_nagnetatelia_newHW;
   ai.Osevoi_sdvig_rotora_nagnetatelia.dLA	    := AI_Osevoi_sdvig_rotora_nagnetatelia_newLA;
   ai.Osevoi_sdvig_rotora_nagnetatelia.dLL	    := AI_Osevoi_sdvig_rotora_nagnetatelia_newLL;
   ai.Osevoi_sdvig_rotora_nagnetatelia.dLW	    := AI_Osevoi_sdvig_rotora_nagnetatelia_newLW;

   ai.Uroven_masla_v_maslobake.inCommand_ARM    := UINT_TO_WORD(AI_Uroven_masla_v_maslobake_command);
   ai.Uroven_masla_v_maslobake.dHL	      := AI_Uroven_masla_v_maslobake_newHL;
   ai.Uroven_masla_v_maslobake.dHW	      := AI_Uroven_masla_v_maslobake_newHW;
   ai.Uroven_masla_v_maslobake.dLA	      := AI_Uroven_masla_v_maslobake_newLA;
   ai.Uroven_masla_v_maslobake.dLL	      := AI_Uroven_masla_v_maslobake_newLL;
   ai.Uroven_masla_v_maslobake.dLW	      := AI_Uroven_masla_v_maslobake_newLW;

  (********************************************* Модуль A1-10 ******************************************************)

   ai.T_vnytri_shkafa.inCommand_ARM	:= UINT_TO_WORD(AI_T_vnytri_shkafa_command);
   ai.T_vnytri_shkafa.dHL    	          := AI_T_vnytri_shkafa_newHL;
   ai.T_vnytri_shkafa.dLL    	          := AI_T_vnytri_shkafa_newLL;
   ai.T_vnytri_shkafa.dHW    	          := AI_T_vnytri_shkafa_newHW;
   ai.T_vnytri_shkafa.dLW    	          := AI_T_vnytri_shkafa_newLW;

   ai.Tok_vozbuzhdeniia_vozbuditelia.inCommand_ARM	:= UINT_TO_WORD(AI_Tok_vozbuzhdeniia_vozbuditelia_command);
   ai.Tok_vozbuzhdeniia_vozbuditelia.dHL    	:= AI_Tok_vozbuzhdeniia_vozbuditelia_newHL;
   ai.Tok_vozbuzhdeniia_vozbuditelia.dLL    	:= AI_Tok_vozbuzhdeniia_vozbuditelia_newLL;

   ai.Tok_statora_elektrodvigatelia.inCommand_ARM	:= UINT_TO_WORD(AI_Tok_statora_elektrodvigatelia_command);
   ai.Tok_statora_elektrodvigatelia.dHL    	:= AI_Tok_statora_elektrodvigatelia_newHL;
   ai.Tok_statora_elektrodvigatelia.dLL    	:= AI_Tok_statora_elektrodvigatelia_newLL;

   ai.Aktivnaia_moshchnost.inCommand_ARM	:= UINT_TO_WORD(AI_Aktivnaia_moshchnost_command);
   ai.Aktivnaia_moshchnost.dHL    	:= AI_Aktivnaia_moshchnost_newHL;
   ai.Aktivnaia_moshchnost.dLL    	:= AI_Aktivnaia_moshchnost_newLL;

   ai.Reaktivnaia_moshchnost.inCommand_ARM	:= UINT_TO_WORD(AI_Reaktivnaia_moshchnost_command);
   ai.Reaktivnaia_moshchnost.dHL            	:= AI_Reaktivnaia_moshchnost_newHL;
   ai.Reaktivnaia_moshchnost.dLL            	:= AI_Reaktivnaia_moshchnost_newLL;

   ai.VoltageSHU_osnovnoi_vvod.inCommand_ARM	:= UINT_TO_WORD(AI_VoltageSHU_osnovnoi_vvod_command);
   ai.VoltageSHU_osnovnoi_vvod.dHL        	:= AI_VoltageSHU_osnovnoi_vvod_newHL;
   ai.VoltageSHU_osnovnoi_vvod.dHW        	:= AI_VoltageSHU_osnovnoi_vvod_newHW;
   ai.VoltageSHU_osnovnoi_vvod.dLL        	:= AI_VoltageSHU_osnovnoi_vvod_newLL;
   ai.VoltageSHU_osnovnoi_vvod.dLW        	:= AI_VoltageSHU_osnovnoi_vvod_newLW;

   ai.VoltageSHU_rezervnyi_vvod.inCommand_ARM	:= UINT_TO_WORD(AI_VoltageSHU_rezervnyi_vvod_command);
   ai.VoltageSHU_rezervnyi_vvod.dHL        	:= AI_VoltageSHU_rezervnyi_vvod_newHL;
   ai.VoltageSHU_rezervnyi_vvod.dHW        	:= AI_VoltageSHU_rezervnyi_vvod_newHW;
   ai.VoltageSHU_rezervnyi_vvod.dLL        	:= AI_VoltageSHU_rezervnyi_vvod_newLL;
   ai.VoltageSHU_rezervnyi_vvod.dLW        	:= AI_VoltageSHU_rezervnyi_vvod_newLW;
END_FUNCTION_BLOCK

FUNCTION_BLOCK OPC_AI_set
  VAR_EXTERNAL
    ai : AiConfig;
    AI_Aktivnaia_moshchnost_HL : LREAL;
    AI_Aktivnaia_moshchnost_LL : LREAL;
    AI_Aktivnaia_moshchnost_command : UINT;
    AI_Aktivnaia_moshchnost_newHL : LREAL;
    AI_Aktivnaia_moshchnost_newLL : LREAL;
    AI_Aktivnaia_moshchnost_status : UDINT;
    AI_Aktivnaia_moshchnost_value : LREAL;
    AI_Osevoi_sdvig_rotora_nagnetatelia_HA : LREAL;
    AI_Osevoi_sdvig_rotora_nagnetatelia_HL : LREAL;
    AI_Osevoi_sdvig_rotora_nagnetatelia_HW : LREAL;
    AI_Osevoi_sdvig_rotora_nagnetatelia_LA : LREAL;
    AI_Osevoi_sdvig_rotora_nagnetatelia_LL : LREAL;
    AI_Osevoi_sdvig_rotora_nagnetatelia_LW : LREAL;
    AI_Osevoi_sdvig_rotora_nagnetatelia_command : UINT;
    AI_Osevoi_sdvig_rotora_nagnetatelia_newHA : LREAL;
    AI_Osevoi_sdvig_rotora_nagnetatelia_newHL : LREAL;
    AI_Osevoi_sdvig_rotora_nagnetatelia_newHW : LREAL;
    AI_Osevoi_sdvig_rotora_nagnetatelia_newLA : LREAL;
    AI_Osevoi_sdvig_rotora_nagnetatelia_newLL : LREAL;
    AI_Osevoi_sdvig_rotora_nagnetatelia_newLW : LREAL;
    AI_Osevoi_sdvig_rotora_nagnetatelia_status : UDINT;
    AI_Osevoi_sdvig_rotora_nagnetatelia_value : LREAL;
    AI_P_gaza_na_vkhode_nagnetatelia_HL : LREAL;
    AI_P_gaza_na_vkhode_nagnetatelia_LL : LREAL;
    AI_P_gaza_na_vkhode_nagnetatelia_command : UINT;
    AI_P_gaza_na_vkhode_nagnetatelia_newHL : LREAL;
    AI_P_gaza_na_vkhode_nagnetatelia_newLL : LREAL;
    AI_P_gaza_na_vkhode_nagnetatelia_status : UDINT;
    AI_P_gaza_na_vkhode_nagnetatelia_value : LREAL;
    AI_P_gaza_na_vykhode_nagnetatelia_HL : LREAL;
    AI_P_gaza_na_vykhode_nagnetatelia_LL : LREAL;
    AI_P_gaza_na_vykhode_nagnetatelia_command : UINT;
    AI_P_gaza_na_vykhode_nagnetatelia_newHL : LREAL;
    AI_P_gaza_na_vykhode_nagnetatelia_newLL : LREAL;
    AI_P_gaza_na_vykhode_nagnetatelia_status : UDINT;
    AI_P_gaza_na_vykhode_nagnetatelia_value : LREAL;
    AI_P_masla_smazki_nizkoe_HL : LREAL;
    AI_P_masla_smazki_nizkoe_LA : LREAL;
    AI_P_masla_smazki_nizkoe_LL : LREAL;
    AI_P_masla_smazki_nizkoe_LW : LREAL;
    AI_P_masla_smazki_nizkoe_command : UINT;
    AI_P_masla_smazki_nizkoe_newHL : LREAL;
    AI_P_masla_smazki_nizkoe_newLA : LREAL;
    AI_P_masla_smazki_nizkoe_newLL : LREAL;
    AI_P_masla_smazki_nizkoe_newLW : LREAL;
    AI_P_masla_smazki_nizkoe_status : UDINT;
    AI_P_masla_smazki_nizkoe_value : LREAL;
    AI_P_masla_smazki_srednee_posle_nasosov_HL : LREAL;
    AI_P_masla_smazki_srednee_posle_nasosov_LL : LREAL;
    AI_P_masla_smazki_srednee_posle_nasosov_LW : LREAL;
    AI_P_masla_smazki_srednee_posle_nasosov_command : UINT;
    AI_P_masla_smazki_srednee_posle_nasosov_newHL : LREAL;
    AI_P_masla_smazki_srednee_posle_nasosov_newLL : LREAL;
    AI_P_masla_smazki_srednee_posle_nasosov_newLW : LREAL;
    AI_P_masla_smazki_srednee_posle_nasosov_status : UDINT;
    AI_P_masla_smazki_srednee_posle_nasosov_value : LREAL;
    AI_P_masla_uplotneniia_HL : LREAL;
    AI_P_masla_uplotneniia_LL : LREAL;
    AI_P_masla_uplotneniia_command : UINT;
    AI_P_masla_uplotneniia_newHL : LREAL;
    AI_P_masla_uplotneniia_newLL : LREAL;
    AI_P_masla_uplotneniia_status : UDINT;
    AI_P_masla_uplotneniia_value : LREAL;
    AI_Reaktivnaia_moshchnost_HL : LREAL;
    AI_Reaktivnaia_moshchnost_LL : LREAL;
    AI_Reaktivnaia_moshchnost_command : UINT;
    AI_Reaktivnaia_moshchnost_newHL : LREAL;
    AI_Reaktivnaia_moshchnost_newLL : LREAL;
    AI_Reaktivnaia_moshchnost_status : UDINT;
    AI_Reaktivnaia_moshchnost_value : LREAL;
    AI_T_aktivnogo_zheleza_statora_1_k_HL : LREAL;
    AI_T_aktivnogo_zheleza_statora_1_k_LL : LREAL;
    AI_T_aktivnogo_zheleza_statora_1_k_command : UINT;
    AI_T_aktivnogo_zheleza_statora_1_k_newHL : LREAL;
    AI_T_aktivnogo_zheleza_statora_1_k_newLL : LREAL;
    AI_T_aktivnogo_zheleza_statora_1_k_status : UDINT;
    AI_T_aktivnogo_zheleza_statora_1_k_value : LREAL;
    AI_T_aktivnogo_zheleza_statora_2_k_HL : LREAL;
    AI_T_aktivnogo_zheleza_statora_2_k_LL : LREAL;
    AI_T_aktivnogo_zheleza_statora_2_k_command : UINT;
    AI_T_aktivnogo_zheleza_statora_2_k_newHL : LREAL;
    AI_T_aktivnogo_zheleza_statora_2_k_newLL : LREAL;
    AI_T_aktivnogo_zheleza_statora_2_k_status : UDINT;
    AI_T_aktivnogo_zheleza_statora_2_k_value : LREAL;
    AI_T_aktivnogo_zheleza_statora_3_k_HL : LREAL;
    AI_T_aktivnogo_zheleza_statora_3_k_LL : LREAL;
    AI_T_aktivnogo_zheleza_statora_3_k_command : UINT;
    AI_T_aktivnogo_zheleza_statora_3_k_newHL : LREAL;
    AI_T_aktivnogo_zheleza_statora_3_k_newLL : LREAL;
    AI_T_aktivnogo_zheleza_statora_3_k_status : UDINT;
    AI_T_aktivnogo_zheleza_statora_3_k_value : LREAL;
    AI_T_clodAir_dvigatelia_t1_HL : LREAL;
    AI_T_clodAir_dvigatelia_t1_LL : LREAL;
    AI_T_clodAir_dvigatelia_t1_command : UINT;
    AI_T_clodAir_dvigatelia_t1_newHL : LREAL;
    AI_T_clodAir_dvigatelia_t1_newLL : LREAL;
    AI_T_clodAir_dvigatelia_t1_status : UDINT;
    AI_T_clodAir_dvigatelia_t1_value : LREAL;
    AI_T_gaz_in_nagnetatelia_HL : LREAL;
    AI_T_gaz_in_nagnetatelia_LL : LREAL;
    AI_T_gaz_in_nagnetatelia_command : UINT;
    AI_T_gaz_in_nagnetatelia_newHL : LREAL;
    AI_T_gaz_in_nagnetatelia_newLL : LREAL;
    AI_T_gaz_in_nagnetatelia_status : UDINT;
    AI_T_gaz_in_nagnetatelia_value : LREAL;
    AI_T_gaz_out_nagnetatelia_HL : LREAL;
    AI_T_gaz_out_nagnetatelia_LL : LREAL;
    AI_T_gaz_out_nagnetatelia_command : UINT;
    AI_T_gaz_out_nagnetatelia_newHL : LREAL;
    AI_T_gaz_out_nagnetatelia_newLL : LREAL;
    AI_T_gaz_out_nagnetatelia_status : UDINT;
    AI_T_gaz_out_nagnetatelia_value : LREAL;
    AI_T_hotAir_dvigatelia_t1_HL : LREAL;
    AI_T_hotAir_dvigatelia_t1_LL : LREAL;
    AI_T_hotAir_dvigatelia_t1_command : UINT;
    AI_T_hotAir_dvigatelia_t1_newHL : LREAL;
    AI_T_hotAir_dvigatelia_t1_newLL : LREAL;
    AI_T_hotAir_dvigatelia_t1_status : UDINT;
    AI_T_hotAir_dvigatelia_t1_value : LREAL;
    AI_T_masla_do_AVOM_HL : LREAL;
    AI_T_masla_do_AVOM_LL : LREAL;
    AI_T_masla_do_AVOM_command : UINT;
    AI_T_masla_do_AVOM_newHL : LREAL;
    AI_T_masla_do_AVOM_newLL : LREAL;
    AI_T_masla_do_AVOM_status : UDINT;
    AI_T_masla_do_AVOM_value : LREAL;
    AI_T_masla_na_slive_perednego_opornogo_podshipnika_dvigatelia_HL : LREAL;
    AI_T_masla_na_slive_perednego_opornogo_podshipnika_dvigatelia_LL : LREAL;
    AI_T_masla_na_slive_perednego_opornogo_podshipnika_dvigatelia_command : UINT;
    AI_T_masla_na_slive_perednego_opornogo_podshipnika_dvigatelia_newHL : LREAL;
    AI_T_masla_na_slive_perednego_opornogo_podshipnika_dvigatelia_newLL : LREAL;
    AI_T_masla_na_slive_perednego_opornogo_podshipnika_dvigatelia_status : UDINT;
    AI_T_masla_na_slive_perednego_opornogo_podshipnika_dvigatelia_value : LREAL;
    AI_T_masla_na_slive_zadnego_opornogo_podshipnika_dvigatelia_HL : LREAL;
    AI_T_masla_na_slive_zadnego_opornogo_podshipnika_dvigatelia_LL : LREAL;
    AI_T_masla_na_slive_zadnego_opornogo_podshipnika_dvigatelia_command : UINT;
    AI_T_masla_na_slive_zadnego_opornogo_podshipnika_dvigatelia_newHL : LREAL;
    AI_T_masla_na_slive_zadnego_opornogo_podshipnika_dvigatelia_newLL : LREAL;
    AI_T_masla_na_slive_zadnego_opornogo_podshipnika_dvigatelia_status : UDINT;
    AI_T_masla_na_slive_zadnego_opornogo_podshipnika_dvigatelia_value : LREAL;
    AI_T_masla_posle_AVOM_HL : LREAL;
    AI_T_masla_posle_AVOM_LL : LREAL;
    AI_T_masla_posle_AVOM_command : UINT;
    AI_T_masla_posle_AVOM_newHL : LREAL;
    AI_T_masla_posle_AVOM_newLL : LREAL;
    AI_T_masla_posle_AVOM_status : UDINT;
    AI_T_masla_posle_AVOM_value : LREAL;
    AI_T_masla_v_maslobake_HL : LREAL;
    AI_T_masla_v_maslobake_HW : LREAL;
    AI_T_masla_v_maslobake_LL : LREAL;
    AI_T_masla_v_maslobake_LW : LREAL;
    AI_T_masla_v_maslobake_command : UINT;
    AI_T_masla_v_maslobake_newHL : LREAL;
    AI_T_masla_v_maslobake_newHW : LREAL;
    AI_T_masla_v_maslobake_newLL : LREAL;
    AI_T_masla_v_maslobake_newLW : LREAL;
    AI_T_masla_v_maslobake_status : UDINT;
    AI_T_masla_v_maslobake_value : LREAL;
    AI_T_obmotki_fazy_1_k_HL : LREAL;
    AI_T_obmotki_fazy_1_k_LL : LREAL;
    AI_T_obmotki_fazy_1_k_command : UINT;
    AI_T_obmotki_fazy_1_k_newHL : LREAL;
    AI_T_obmotki_fazy_1_k_newLL : LREAL;
    AI_T_obmotki_fazy_1_k_status : UDINT;
    AI_T_obmotki_fazy_1_k_value : LREAL;
    AI_T_obmotki_fazy_2_k_HL : LREAL;
    AI_T_obmotki_fazy_2_k_LL : LREAL;
    AI_T_obmotki_fazy_2_k_command : UINT;
    AI_T_obmotki_fazy_2_k_newHL : LREAL;
    AI_T_obmotki_fazy_2_k_newLL : LREAL;
    AI_T_obmotki_fazy_2_k_status : UDINT;
    AI_T_obmotki_fazy_2_k_value : LREAL;
    AI_T_obmotki_fazy_3_k_HL : LREAL;
    AI_T_obmotki_fazy_3_k_LL : LREAL;
    AI_T_obmotki_fazy_3_k_command : UINT;
    AI_T_obmotki_fazy_3_k_newHL : LREAL;
    AI_T_obmotki_fazy_3_k_newLL : LREAL;
    AI_T_obmotki_fazy_3_k_status : UDINT;
    AI_T_obmotki_fazy_3_k_value : LREAL;
    AI_T_oporno_upornogo_podshipnika_nagnetatelia_t4_HA : LREAL;
    AI_T_oporno_upornogo_podshipnika_nagnetatelia_t4_HL : LREAL;
    AI_T_oporno_upornogo_podshipnika_nagnetatelia_t4_HW : LREAL;
    AI_T_oporno_upornogo_podshipnika_nagnetatelia_t4_LL : LREAL;
    AI_T_oporno_upornogo_podshipnika_nagnetatelia_t4_command : UINT;
    AI_T_oporno_upornogo_podshipnika_nagnetatelia_t4_newHA : LREAL;
    AI_T_oporno_upornogo_podshipnika_nagnetatelia_t4_newHL : LREAL;
    AI_T_oporno_upornogo_podshipnika_nagnetatelia_t4_newHW : LREAL;
    AI_T_oporno_upornogo_podshipnika_nagnetatelia_t4_newLL : LREAL;
    AI_T_oporno_upornogo_podshipnika_nagnetatelia_t4_status : UDINT;
    AI_T_oporno_upornogo_podshipnika_nagnetatelia_t4_value : LREAL;
    AI_T_opornogo_podshipnika_nagnetatelia_t1_HA : LREAL;
    AI_T_opornogo_podshipnika_nagnetatelia_t1_HL : LREAL;
    AI_T_opornogo_podshipnika_nagnetatelia_t1_HW : LREAL;
    AI_T_opornogo_podshipnika_nagnetatelia_t1_LL : LREAL;
    AI_T_opornogo_podshipnika_nagnetatelia_t1_command : UINT;
    AI_T_opornogo_podshipnika_nagnetatelia_t1_newHA : LREAL;
    AI_T_opornogo_podshipnika_nagnetatelia_t1_newHL : LREAL;
    AI_T_opornogo_podshipnika_nagnetatelia_t1_newHW : LREAL;
    AI_T_opornogo_podshipnika_nagnetatelia_t1_newLL : LREAL;
    AI_T_opornogo_podshipnika_nagnetatelia_t1_status : UDINT;
    AI_T_opornogo_podshipnika_nagnetatelia_t1_value : LREAL;
    AI_T_opornogo_podshipnika_nagnetatelia_t2_HA : LREAL;
    AI_T_opornogo_podshipnika_nagnetatelia_t2_HL : LREAL;
    AI_T_opornogo_podshipnika_nagnetatelia_t2_HW : LREAL;
    AI_T_opornogo_podshipnika_nagnetatelia_t2_LL : LREAL;
    AI_T_opornogo_podshipnika_nagnetatelia_t2_command : UINT;
    AI_T_opornogo_podshipnika_nagnetatelia_t2_newHA : LREAL;
    AI_T_opornogo_podshipnika_nagnetatelia_t2_newHL : LREAL;
    AI_T_opornogo_podshipnika_nagnetatelia_t2_newHW : LREAL;
    AI_T_opornogo_podshipnika_nagnetatelia_t2_newLL : LREAL;
    AI_T_opornogo_podshipnika_nagnetatelia_t2_status : UDINT;
    AI_T_opornogo_podshipnika_nagnetatelia_t2_value : LREAL;
    AI_T_opornogo_podshipnika_nagnetatelia_t3_HA : LREAL;
    AI_T_opornogo_podshipnika_nagnetatelia_t3_HL : LREAL;
    AI_T_opornogo_podshipnika_nagnetatelia_t3_HW : LREAL;
    AI_T_opornogo_podshipnika_nagnetatelia_t3_LL : LREAL;
    AI_T_opornogo_podshipnika_nagnetatelia_t3_command : UINT;
    AI_T_opornogo_podshipnika_nagnetatelia_t3_newHA : LREAL;
    AI_T_opornogo_podshipnika_nagnetatelia_t3_newHL : LREAL;
    AI_T_opornogo_podshipnika_nagnetatelia_t3_newHW : LREAL;
    AI_T_opornogo_podshipnika_nagnetatelia_t3_newLL : LREAL;
    AI_T_opornogo_podshipnika_nagnetatelia_t3_status : UDINT;
    AI_T_opornogo_podshipnika_nagnetatelia_t3_value : LREAL;
    AI_T_perednego_opornogo_podshipnika_dvigatelia_t1_HL : LREAL;
    AI_T_perednego_opornogo_podshipnika_dvigatelia_t1_LL : LREAL;
    AI_T_perednego_opornogo_podshipnika_dvigatelia_t1_command : UINT;
    AI_T_perednego_opornogo_podshipnika_dvigatelia_t1_newHL : LREAL;
    AI_T_perednego_opornogo_podshipnika_dvigatelia_t1_newLL : LREAL;
    AI_T_perednego_opornogo_podshipnika_dvigatelia_t1_status : UDINT;
    AI_T_perednego_opornogo_podshipnika_dvigatelia_t1_value : LREAL;
    AI_T_podshipnika_reduktora_t1_HA : LREAL;
    AI_T_podshipnika_reduktora_t1_HL : LREAL;
    AI_T_podshipnika_reduktora_t1_HW : LREAL;
    AI_T_podshipnika_reduktora_t1_LL : LREAL;
    AI_T_podshipnika_reduktora_t1_command : UINT;
    AI_T_podshipnika_reduktora_t1_newHA : LREAL;
    AI_T_podshipnika_reduktora_t1_newHL : LREAL;
    AI_T_podshipnika_reduktora_t1_newHW : LREAL;
    AI_T_podshipnika_reduktora_t1_newLL : LREAL;
    AI_T_podshipnika_reduktora_t1_status : UDINT;
    AI_T_podshipnika_reduktora_t1_value : LREAL;
    AI_T_podshipnika_reduktora_t2_HA : LREAL;
    AI_T_podshipnika_reduktora_t2_HL : LREAL;
    AI_T_podshipnika_reduktora_t2_HW : LREAL;
    AI_T_podshipnika_reduktora_t2_LL : LREAL;
    AI_T_podshipnika_reduktora_t2_command : UINT;
    AI_T_podshipnika_reduktora_t2_newHA : LREAL;
    AI_T_podshipnika_reduktora_t2_newHL : LREAL;
    AI_T_podshipnika_reduktora_t2_newHW : LREAL;
    AI_T_podshipnika_reduktora_t2_newLL : LREAL;
    AI_T_podshipnika_reduktora_t2_status : UDINT;
    AI_T_podshipnika_reduktora_t2_value : LREAL;
    AI_T_podshipnika_reduktora_t3_HA : LREAL;
    AI_T_podshipnika_reduktora_t3_HL : LREAL;
    AI_T_podshipnika_reduktora_t3_HW : LREAL;
    AI_T_podshipnika_reduktora_t3_LL : LREAL;
    AI_T_podshipnika_reduktora_t3_command : UINT;
    AI_T_podshipnika_reduktora_t3_newHA : LREAL;
    AI_T_podshipnika_reduktora_t3_newHL : LREAL;
    AI_T_podshipnika_reduktora_t3_newHW : LREAL;
    AI_T_podshipnika_reduktora_t3_newLL : LREAL;
    AI_T_podshipnika_reduktora_t3_status : UDINT;
    AI_T_podshipnika_reduktora_t3_value : LREAL;
    AI_T_podshipnika_reduktora_t4_HA : LREAL;
    AI_T_podshipnika_reduktora_t4_HL : LREAL;
    AI_T_podshipnika_reduktora_t4_HW : LREAL;
    AI_T_podshipnika_reduktora_t4_LL : LREAL;
    AI_T_podshipnika_reduktora_t4_command : UINT;
    AI_T_podshipnika_reduktora_t4_newHA : LREAL;
    AI_T_podshipnika_reduktora_t4_newHL : LREAL;
    AI_T_podshipnika_reduktora_t4_newHW : LREAL;
    AI_T_podshipnika_reduktora_t4_newLL : LREAL;
    AI_T_podshipnika_reduktora_t4_status : UDINT;
    AI_T_podshipnika_reduktora_t4_value : LREAL;
    AI_T_zadnego_opornogo_podshipnika_dvigatelia_t2_HA : LREAL;
    AI_T_zadnego_opornogo_podshipnika_dvigatelia_t2_HL : LREAL;
    AI_T_zadnego_opornogo_podshipnika_dvigatelia_t2_HW : LREAL;
    AI_T_zadnego_opornogo_podshipnika_dvigatelia_t2_LL : LREAL;
    AI_T_zadnego_opornogo_podshipnika_dvigatelia_t2_command : UINT;
    AI_T_zadnego_opornogo_podshipnika_dvigatelia_t2_newHA : LREAL;
    AI_T_zadnego_opornogo_podshipnika_dvigatelia_t2_newHL : LREAL;
    AI_T_zadnego_opornogo_podshipnika_dvigatelia_t2_newHW : LREAL;
    AI_T_zadnego_opornogo_podshipnika_dvigatelia_t2_newLL : LREAL;
    AI_T_zadnego_opornogo_podshipnika_dvigatelia_t2_status : UDINT;
    AI_T_zadnego_opornogo_podshipnika_dvigatelia_t2_value : LREAL;
    AI_Tok_statora_elektrodvigatelia_HL : LREAL;
    AI_Tok_statora_elektrodvigatelia_LL : LREAL;
    AI_Tok_statora_elektrodvigatelia_command : UINT;
    AI_Tok_statora_elektrodvigatelia_newHL : LREAL;
    AI_Tok_statora_elektrodvigatelia_newLL : LREAL;
    AI_Tok_statora_elektrodvigatelia_status : UDINT;
    AI_Tok_statora_elektrodvigatelia_value : LREAL;
    AI_Tok_vozbuzhdeniia_vozbuditelia_HL : LREAL;
    AI_Tok_vozbuzhdeniia_vozbuditelia_LL : LREAL;
    AI_Tok_vozbuzhdeniia_vozbuditelia_command : UINT;
    AI_Tok_vozbuzhdeniia_vozbuditelia_newHL : LREAL;
    AI_Tok_vozbuzhdeniia_vozbuditelia_newLL : LREAL;
    AI_Tok_vozbuzhdeniia_vozbuditelia_status : UDINT;
    AI_Tok_vozbuzhdeniia_vozbuditelia_value : LREAL;
    AI_Uroven_masla_v_maslobake_HL : LREAL;
    AI_Uroven_masla_v_maslobake_HW : LREAL;
    AI_Uroven_masla_v_maslobake_LA : LREAL;
    AI_Uroven_masla_v_maslobake_LL : LREAL;
    AI_Uroven_masla_v_maslobake_LW : LREAL;
    AI_Uroven_masla_v_maslobake_command : UINT;
    AI_Uroven_masla_v_maslobake_newHL : LREAL;
    AI_Uroven_masla_v_maslobake_newHW : LREAL;
    AI_Uroven_masla_v_maslobake_newLA : LREAL;
    AI_Uroven_masla_v_maslobake_newLL : LREAL;
    AI_Uroven_masla_v_maslobake_newLW : LREAL;
    AI_Uroven_masla_v_maslobake_status : UDINT;
    AI_Uroven_masla_v_maslobake_value : LREAL;
    AI_Vibratciia_STD_t1_HA : LREAL;
    AI_Vibratciia_STD_t1_HL : LREAL;
    AI_Vibratciia_STD_t1_HW : LREAL;
    AI_Vibratciia_STD_t1_LL : LREAL;
    AI_Vibratciia_STD_t1_command : UINT;
    AI_Vibratciia_STD_t1_newHA : LREAL;
    AI_Vibratciia_STD_t1_newHL : LREAL;
    AI_Vibratciia_STD_t1_newHW : LREAL;
    AI_Vibratciia_STD_t1_newLL : LREAL;
    AI_Vibratciia_STD_t1_status : UDINT;
    AI_Vibratciia_STD_t1_value : LREAL;
    AI_Vibratciia_STD_t2_HA : LREAL;
    AI_Vibratciia_STD_t2_HL : LREAL;
    AI_Vibratciia_STD_t2_HW : LREAL;
    AI_Vibratciia_STD_t2_LL : LREAL;
    AI_Vibratciia_STD_t2_command : UINT;
    AI_Vibratciia_STD_t2_newHA : LREAL;
    AI_Vibratciia_STD_t2_newHL : LREAL;
    AI_Vibratciia_STD_t2_newHW : LREAL;
    AI_Vibratciia_STD_t2_newLL : LREAL;
    AI_Vibratciia_STD_t2_status : UDINT;
    AI_Vibratciia_STD_t2_value : LREAL;
    AI_Vibratciia_rotora_nagnetatelia_t1_HA : LREAL;
    AI_Vibratciia_rotora_nagnetatelia_t1_HL : LREAL;
    AI_Vibratciia_rotora_nagnetatelia_t1_HW : LREAL;
    AI_Vibratciia_rotora_nagnetatelia_t1_LL : LREAL;
    AI_Vibratciia_rotora_nagnetatelia_t1_command : UINT;
    AI_Vibratciia_rotora_nagnetatelia_t1_newHA : LREAL;
    AI_Vibratciia_rotora_nagnetatelia_t1_newHL : LREAL;
    AI_Vibratciia_rotora_nagnetatelia_t1_newHW : LREAL;
    AI_Vibratciia_rotora_nagnetatelia_t1_newLL : LREAL;
    AI_Vibratciia_rotora_nagnetatelia_t1_status : UDINT;
    AI_Vibratciia_rotora_nagnetatelia_t1_value : LREAL;
    AI_Vibratciia_rotora_nagnetatelia_t2_HA : LREAL;
    AI_Vibratciia_rotora_nagnetatelia_t2_HL : LREAL;
    AI_Vibratciia_rotora_nagnetatelia_t2_HW : LREAL;
    AI_Vibratciia_rotora_nagnetatelia_t2_LL : LREAL;
    AI_Vibratciia_rotora_nagnetatelia_t2_command : UINT;
    AI_Vibratciia_rotora_nagnetatelia_t2_newHA : LREAL;
    AI_Vibratciia_rotora_nagnetatelia_t2_newHL : LREAL;
    AI_Vibratciia_rotora_nagnetatelia_t2_newHW : LREAL;
    AI_Vibratciia_rotora_nagnetatelia_t2_newLL : LREAL;
    AI_Vibratciia_rotora_nagnetatelia_t2_status : UDINT;
    AI_Vibratciia_rotora_nagnetatelia_t2_value : LREAL;
    AI_Vibratciia_rotora_nagnetatelia_t3_HA : LREAL;
    AI_Vibratciia_rotora_nagnetatelia_t3_HL : LREAL;
    AI_Vibratciia_rotora_nagnetatelia_t3_HW : LREAL;
    AI_Vibratciia_rotora_nagnetatelia_t3_LL : LREAL;
    AI_Vibratciia_rotora_nagnetatelia_t3_command : UINT;
    AI_Vibratciia_rotora_nagnetatelia_t3_newHA : LREAL;
    AI_Vibratciia_rotora_nagnetatelia_t3_newHL : LREAL;
    AI_Vibratciia_rotora_nagnetatelia_t3_newHW : LREAL;
    AI_Vibratciia_rotora_nagnetatelia_t3_newLL : LREAL;
    AI_Vibratciia_rotora_nagnetatelia_t3_status : UDINT;
    AI_Vibratciia_rotora_nagnetatelia_t3_value : LREAL;
    AI_Vibratciia_rotora_nagnetatelia_t4_HA : LREAL;
    AI_Vibratciia_rotora_nagnetatelia_t4_HL : LREAL;
    AI_Vibratciia_rotora_nagnetatelia_t4_HW : LREAL;
    AI_Vibratciia_rotora_nagnetatelia_t4_LL : LREAL;
    AI_Vibratciia_rotora_nagnetatelia_t4_command : UINT;
    AI_Vibratciia_rotora_nagnetatelia_t4_newHA : LREAL;
    AI_Vibratciia_rotora_nagnetatelia_t4_newHL : LREAL;
    AI_Vibratciia_rotora_nagnetatelia_t4_newHW : LREAL;
    AI_Vibratciia_rotora_nagnetatelia_t4_newLL : LREAL;
    AI_Vibratciia_rotora_nagnetatelia_t4_status : UDINT;
    AI_Vibratciia_rotora_nagnetatelia_t4_value : LREAL;
    AI_VoltageSHU_osnovnoi_vvod_HL : LREAL;
    AI_VoltageSHU_osnovnoi_vvod_HW : LREAL;
    AI_VoltageSHU_osnovnoi_vvod_LL : LREAL;
    AI_VoltageSHU_osnovnoi_vvod_LW : LREAL;
    AI_VoltageSHU_osnovnoi_vvod_command : UINT;
    AI_VoltageSHU_osnovnoi_vvod_newHL : LREAL;
    AI_VoltageSHU_osnovnoi_vvod_newHW : LREAL;
    AI_VoltageSHU_osnovnoi_vvod_newLL : LREAL;
    AI_VoltageSHU_osnovnoi_vvod_newLW : LREAL;
    AI_VoltageSHU_osnovnoi_vvod_status : UDINT;
    AI_VoltageSHU_osnovnoi_vvod_value : LREAL;
    AI_VoltageSHU_rezervnyi_vvod_HL : LREAL;
    AI_VoltageSHU_rezervnyi_vvod_HW : LREAL;
    AI_VoltageSHU_rezervnyi_vvod_LL : LREAL;
    AI_VoltageSHU_rezervnyi_vvod_LW : LREAL;
    AI_VoltageSHU_rezervnyi_vvod_command : UINT;
    AI_VoltageSHU_rezervnyi_vvod_newHL : LREAL;
    AI_VoltageSHU_rezervnyi_vvod_newHW : LREAL;
    AI_VoltageSHU_rezervnyi_vvod_newLL : LREAL;
    AI_VoltageSHU_rezervnyi_vvod_newLW : LREAL;
    AI_VoltageSHU_rezervnyi_vvod_status : UDINT;
    AI_VoltageSHU_rezervnyi_vvod_value : LREAL;
    AI_dP_gaza_na_konfuzore_nagnetatelia_HL : LREAL;
    AI_dP_gaza_na_konfuzore_nagnetatelia_LL : LREAL;
    AI_dP_gaza_na_konfuzore_nagnetatelia_command : UINT;
    AI_dP_gaza_na_konfuzore_nagnetatelia_newHL : LREAL;
    AI_dP_gaza_na_konfuzore_nagnetatelia_newLL : LREAL;
    AI_dP_gaza_na_konfuzore_nagnetatelia_status : UDINT;
    AI_dP_gaza_na_konfuzore_nagnetatelia_value : LREAL;
    AI_dPmaslo_gaz_HL : LREAL;
    AI_dPmaslo_gaz_LA : LREAL;
    AI_dPmaslo_gaz_LL : LREAL;
    AI_dPmaslo_gaz_LW : LREAL;
    AI_dPmaslo_gaz_command : UINT;
    AI_dPmaslo_gaz_newHL : LREAL;
    AI_dPmaslo_gaz_newLA : LREAL;
    AI_dPmaslo_gaz_newLL : LREAL;
    AI_dPmaslo_gaz_newLW : LREAL;
    AI_dPmaslo_gaz_status : UDINT;
    AI_dPmaslo_gaz_value : LREAL;
    AI_T_perednego_opornogo_podshipnika_dvigatelia_t1_HA : LREAL;
    AI_T_perednego_opornogo_podshipnika_dvigatelia_t1_HW : LREAL;
    AI_T_perednego_opornogo_podshipnika_dvigatelia_t1_newHA : LREAL;
    AI_T_perednego_opornogo_podshipnika_dvigatelia_t1_newHW : LREAL;
    AI_T_gaz_out_nagnetatelia_HA : LREAL;
    AI_T_gaz_out_nagnetatelia_HW : LREAL;
    AI_T_gaz_out_nagnetatelia_newHA : LREAL;
    AI_T_gaz_out_nagnetatelia_newHW : LREAL;
    algoritms_AntiPompag_q_Value : LREAL;
    algoritms_AntiPompag_q_status : UDINT;
    algoritms_AntiPompag_zapas_Value : LREAL;
    algoritms_AntiPompag_zapas_status : UDINT;
    AI_T_vnytri_shkafa_HL : LREAL;
    AI_T_vnytri_shkafa_HW : LREAL;
    AI_T_vnytri_shkafa_LL : LREAL;
    AI_T_vnytri_shkafa_LW : LREAL;
    AI_T_vnytri_shkafa_status : UDINT;
    AI_T_vnytri_shkafa_value : LREAL;
    AI_dPmaslo_gaz_MaxChangeDown : LREAL;
    AI_dPmaslo_gaz_MaxChangeUP : LREAL;
  END_VAR

  (* OPC Set - AI. Запись текущих состояний тэгов _______________________________________________________*)

  (********************************************* Модуль A1-4 ******************************************************)

  AI_T_obmotki_fazy_1_k_HL       := ai.T_obmotki_fazy_1_k.HL;
  AI_T_obmotki_fazy_1_k_LL       := ai.T_obmotki_fazy_1_k.LL;
  AI_T_obmotki_fazy_1_k_status := DWORD_TO_UDINT(ai.T_obmotki_fazy_1_k.status);
  AI_T_obmotki_fazy_1_k_value := ai.T_obmotki_fazy_1_k.value;

  AI_T_aktivnogo_zheleza_statora_1_k_HL        := ai.T_aktivnogo_zheleza_statora_1_k.HL;
  AI_T_aktivnogo_zheleza_statora_1_k_LL        := ai.T_aktivnogo_zheleza_statora_1_k.LL;
  AI_T_aktivnogo_zheleza_statora_1_k_status := DWORD_TO_UDINT(ai.T_aktivnogo_zheleza_statora_1_k.status);
  AI_T_aktivnogo_zheleza_statora_1_k_value := ai.T_aktivnogo_zheleza_statora_1_k.value;

  AI_T_obmotki_fazy_2_k_HL	:= ai.T_obmotki_fazy_2_k.HL;
  AI_T_obmotki_fazy_2_k_LL	:= ai.T_obmotki_fazy_2_k.LL;
  AI_T_obmotki_fazy_2_k_status := DWORD_TO_UDINT(ai.T_obmotki_fazy_2_k.status);
  AI_T_obmotki_fazy_2_k_value := ai.T_obmotki_fazy_2_k.value;

  AI_T_aktivnogo_zheleza_statora_2_k_HL       := ai.T_aktivnogo_zheleza_statora_2_k.HL;
  AI_T_aktivnogo_zheleza_statora_2_k_LL       := ai.T_aktivnogo_zheleza_statora_2_k.LL;
  AI_T_aktivnogo_zheleza_statora_2_k_status := DWORD_TO_UDINT(ai.T_aktivnogo_zheleza_statora_2_k.status);
  AI_T_aktivnogo_zheleza_statora_2_k_value := ai.T_aktivnogo_zheleza_statora_2_k.value;

  AI_T_obmotki_fazy_3_k_HL	:= ai.T_obmotki_fazy_3_k.HL;
  AI_T_obmotki_fazy_3_k_LL	:= ai.T_obmotki_fazy_3_k.LL;
  AI_T_obmotki_fazy_3_k_status := DWORD_TO_UDINT(ai.T_obmotki_fazy_3_k.status);
  AI_T_obmotki_fazy_3_k_value := ai.T_obmotki_fazy_3_k.value;

  AI_T_aktivnogo_zheleza_statora_3_k_HL	    := ai.T_aktivnogo_zheleza_statora_3_k.HL;
  AI_T_aktivnogo_zheleza_statora_3_k_LL	    := ai.T_aktivnogo_zheleza_statora_3_k.LL;
  AI_T_aktivnogo_zheleza_statora_3_k_status := DWORD_TO_UDINT(ai.T_aktivnogo_zheleza_statora_3_k.status);
  AI_T_aktivnogo_zheleza_statora_3_k_value := ai.T_aktivnogo_zheleza_statora_3_k.value;

  AI_T_masla_v_maslobake_HL	:= ai.T_masla_v_maslobake.HL;
  AI_T_masla_v_maslobake_HW	:= ai.T_masla_v_maslobake.HW;
  AI_T_masla_v_maslobake_LL	:= ai.T_masla_v_maslobake.LL;
  AI_T_masla_v_maslobake_LW	:= ai.T_masla_v_maslobake.LW;
  AI_T_masla_v_maslobake_status := DWORD_TO_UDINT(ai.T_masla_v_maslobake.status);
  AI_T_masla_v_maslobake_value := ai.T_masla_v_maslobake.value;

  (********************************************* Модуль A1-5 ******************************************************)
  AI_T_perednego_opornogo_podshipnika_dvigatelia_t1_HA	:= ai.T_perednego_opornogo_podshipnika_dvigatelia_t1.HA;
  AI_T_perednego_opornogo_podshipnika_dvigatelia_t1_HL	:= ai.T_perednego_opornogo_podshipnika_dvigatelia_t1.HL;
  AI_T_perednego_opornogo_podshipnika_dvigatelia_t1_HW	:= ai.T_perednego_opornogo_podshipnika_dvigatelia_t1.HW;
  AI_T_perednego_opornogo_podshipnika_dvigatelia_t1_LL	:= ai.T_perednego_opornogo_podshipnika_dvigatelia_t1.LL;
  AI_T_perednego_opornogo_podshipnika_dvigatelia_t1_status := DWORD_TO_UDINT(ai.T_perednego_opornogo_podshipnika_dvigatelia_t1.status);
  AI_T_perednego_opornogo_podshipnika_dvigatelia_t1_value := ai.T_perednego_opornogo_podshipnika_dvigatelia_t1.value;

  AI_T_zadnego_opornogo_podshipnika_dvigatelia_t2_HA	:= ai.T_zadnego_opornogo_podshipnika_dvigatelia_t2.HA;
  AI_T_zadnego_opornogo_podshipnika_dvigatelia_t2_HL	:= ai.T_zadnego_opornogo_podshipnika_dvigatelia_t2.HL;
  AI_T_zadnego_opornogo_podshipnika_dvigatelia_t2_HW	:= ai.T_zadnego_opornogo_podshipnika_dvigatelia_t2.HW;
  AI_T_zadnego_opornogo_podshipnika_dvigatelia_t2_LL	:= ai.T_zadnego_opornogo_podshipnika_dvigatelia_t2.LL;
  AI_T_zadnego_opornogo_podshipnika_dvigatelia_t2_status := DWORD_TO_UDINT(ai.T_zadnego_opornogo_podshipnika_dvigatelia_t2.status);
  AI_T_zadnego_opornogo_podshipnika_dvigatelia_t2_value := ai.T_zadnego_opornogo_podshipnika_dvigatelia_t2.value;

  AI_T_masla_na_slive_perednego_opornogo_podshipnika_dvigatelia_HL	:= ai.T_masla_na_slive_perednego_opornogo_podshipnika_dvigatelia.HL;
  AI_T_masla_na_slive_perednego_opornogo_podshipnika_dvigatelia_LL	:= ai.T_masla_na_slive_perednego_opornogo_podshipnika_dvigatelia.LL;
  AI_T_masla_na_slive_perednego_opornogo_podshipnika_dvigatelia_status := DWORD_TO_UDINT(ai.T_masla_na_slive_perednego_opornogo_podshipnika_dvigatelia.status);
  AI_T_masla_na_slive_perednego_opornogo_podshipnika_dvigatelia_value := ai.T_masla_na_slive_perednego_opornogo_podshipnika_dvigatelia.value;

  AI_T_masla_na_slive_zadnego_opornogo_podshipnika_dvigatelia_HL	:= ai.T_masla_na_slive_zadnego_opornogo_podshipnika_dvigatelia.HL;
  AI_T_masla_na_slive_zadnego_opornogo_podshipnika_dvigatelia_LL	:= ai.T_masla_na_slive_zadnego_opornogo_podshipnika_dvigatelia.LL;
  AI_T_masla_na_slive_zadnego_opornogo_podshipnika_dvigatelia_status := DWORD_TO_UDINT(ai.T_masla_na_slive_zadnego_opornogo_podshipnika_dvigatelia.status);
  AI_T_masla_na_slive_zadnego_opornogo_podshipnika_dvigatelia_value := ai.T_masla_na_slive_zadnego_opornogo_podshipnika_dvigatelia.value;

  AI_T_podshipnika_reduktora_t1_HA	:= ai.T_podshipnika_reduktora_t1.HA;
  AI_T_podshipnika_reduktora_t1_HL	:= ai.T_podshipnika_reduktora_t1.HL;
  AI_T_podshipnika_reduktora_t1_HW	:= ai.T_podshipnika_reduktora_t1.HW;
  AI_T_podshipnika_reduktora_t1_LL	:= ai.T_podshipnika_reduktora_t1.LL;
  AI_T_podshipnika_reduktora_t1_status := DWORD_TO_UDINT(ai.T_podshipnika_reduktora_t1.status);
  AI_T_podshipnika_reduktora_t1_value := ai.T_podshipnika_reduktora_t1.value;

  AI_T_podshipnika_reduktora_t2_HA	:= ai.T_podshipnika_reduktora_t2.HA;
  AI_T_podshipnika_reduktora_t2_HL	:= ai.T_podshipnika_reduktora_t2.HL;
  AI_T_podshipnika_reduktora_t2_HW	:= ai.T_podshipnika_reduktora_t2.HW;
  AI_T_podshipnika_reduktora_t2_LL	:= ai.T_podshipnika_reduktora_t2.LL;
  AI_T_podshipnika_reduktora_t2_status := DWORD_TO_UDINT(ai.T_podshipnika_reduktora_t2.status);
  AI_T_podshipnika_reduktora_t2_value := ai.T_podshipnika_reduktora_t2.value;

  AI_T_podshipnika_reduktora_t3_HA	:= ai.T_podshipnika_reduktora_t3.HA;
  AI_T_podshipnika_reduktora_t3_HL	:= ai.T_podshipnika_reduktora_t3.HL;
  AI_T_podshipnika_reduktora_t3_HW	:= ai.T_podshipnika_reduktora_t3.HW;
  AI_T_podshipnika_reduktora_t3_LL	:= ai.T_podshipnika_reduktora_t3.LL;
  AI_T_podshipnika_reduktora_t3_status := DWORD_TO_UDINT(ai.T_podshipnika_reduktora_t3.status);
  AI_T_podshipnika_reduktora_t3_value := ai.T_podshipnika_reduktora_t3.value;

  AI_T_podshipnika_reduktora_t4_HA	:= ai.T_podshipnika_reduktora_t4.HA;
  AI_T_podshipnika_reduktora_t4_HL	:= ai.T_podshipnika_reduktora_t4.HL;
  AI_T_podshipnika_reduktora_t4_HW	:= ai.T_podshipnika_reduktora_t4.HW;
  AI_T_podshipnika_reduktora_t4_LL	:= ai.T_podshipnika_reduktora_t4.LL;
  AI_T_podshipnika_reduktora_t4_status := DWORD_TO_UDINT(ai.T_podshipnika_reduktora_t4.status);
  AI_T_podshipnika_reduktora_t4_value := ai.T_podshipnika_reduktora_t4.value;
